LIN {X 0,Y 274.627,Z 437.441,A -85,B 0,C 180,E1 -17711.091,E2 -17711.091} C_VEL
LIN {X 0,Y 272.155,Z 443.733,A -85,B 0,C 180,E1 -17713.497,E2 -17713.497} C_VEL
LIN {X 0,Y 270.137,Z 449.54,A -85,B 0,C 180,E1 -17716.459,E2 -17716.459} C_VEL
LIN {X 0,Y 269.337,Z 451.749,A -85,B 0,C 180,E1 -17717.951,E2 -17717.951} C_VEL
LIN {X 0,Y 268.643,Z 455.017,A -85,B 0,C 180,E1 -17720.969,E2 -17720.969} C_VEL
LIN {X 0,Y 268.592,Z 456.649,A -85,B 0,C 180,E1 -17723.992,E2 -17723.992} C_VEL
LIN {X 0,Y 268.676,Z 456.883,A -85,B 0,C 180,E1 -17725.499,E2 -17725.499} C_VEL
LIN {X 0,Y 268.958,Z 456.687,A -85,B 0,C 180,E1 -17727.004,E2 -17727.004} C_VEL
LIN {X 0,Y 269.249,Z 456.062,A -85,B 0,C 180,E1 -17728.504,E2 -17728.504} C_VEL
LIN {X 0,Y 269.5,Z 453.773,A -85,B 0,C 180,E1 -17731.214,E2 -17731.214} C_VEL
LIN {X 0,Y 269.104,Z 455.004,A -85,B 0,C 180,E1 -17732.994,E2 -17732.994} C_VEL
LIN {X 0,Y 268.764,Z 455.392,A -85,B 0,C 180,E1 -17734.499,E2 -17734.499} C_VEL
LIN {X 0,Y 268.716,Z 454.986,A -85,B 0,C 180,E1 -17736.344,E2 -17736.344} C_VEL
LIN {X 0,Y 268.741,Z 454.264,A -85,B 0,C 180,E1 -17737.513,E2 -17737.513} C_VEL
LIN {X 0,Y 269.089,Z 451.749,A -85,B 0,C 180,E1 -17739.774,E2 -17739.774} C_VEL
LIN {X 0,Y 269.857,Z 447.728,A -85,B 0,C 180,E1 -17742.026,E2 -17742.026} C_VEL
LIN {X 0,Y 270.951,Z 443.145,A -85,B 0,C 180,E1 -17743.882,E2 -17743.882} C_VEL
LIN {X 0,Y 272.382,Z 437.177,A -85,B 0,C 180,E1 -17745.719,E2 -17745.719} C_VEL
LIN {X 0,Y 274.136,Z 429.673,A -85,B 0,C 180,E1 -17747.532,E2 -17747.532} C_VEL
LIN {X 0,Y 276.003,Z 420.924,A -85,B 0,C 180,E1 -17749.133,E2 -17749.133} C_VEL
LIN {X 0,Y 277.817,Z 411.718,A -85,B 0,C 180,E1 -17750.439,E2 -17750.439} C_VEL
LIN {X 0,Y 278.918,Z 404.593,A -85,B 0,C 180,E1 -17751.255,E2 -17751.255} C_VEL
LIN {X 0,Y 278.981,Z 396.262,A -85,B 0,C 180,E1 -17752.202,E2 -17752.202} C_VEL
LIN {X 0,Y 278.566,Z 384.711,A -85,B 0,C 180,E1 -17753.315,E2 -17753.315} C_VEL
LIN {X 0,Y 278.989,Z 376.477,A -85,B 0,C 180,E1 -17755.047,E2 -17755.047} C_VEL
LIN {X 0,Y 279.925,Z 365.219,A -85,B 0,C 180,E1 -17757.799,E2 -17757.799} C_VEL
LIN {X 0,Y 281.461,Z 354.384,A -85,B 0,C 180,E1 -17761.019,E2 -17761.019} C_VEL
LIN {X 0,Y 282.099,Z 351.247,A -85,B 0,C 180,E1 -17762.105,E2 -17762.105} C_VEL
LIN {X 0,Y 282.162,Z 348.83,A -85,B 0,C 180,E1 -17763.228,E2 -17763.228} C_VEL
LIN {X 0,Y 281.757,Z 343.357,A -85,B 0,C 180,E1 -17766.773,E2 -17766.773} C_VEL
LIN {X 0,Y 281.788,Z 340.66,A -85,B 0,C 180,E1 -17769.359,E2 -17769.359} C_VEL
LIN {X 0,Y 281.455,Z 339.512,A -85,B 0,C 180,E1 -17771.485,E2 -17771.485} C_VEL
LIN {X 0,Y 280.869,Z 339.07,A -85,B 0,C 180,E1 -17774.477,E2 -17774.477} C_VEL
LIN {X 0,Y 280.547,Z 339.568,A -85,B 0,C 180,E1 -17777.437,E2 -17777.437} C_VEL
LIN {X 0,Y 280.361,Z 341.176,A -85,B 0,C 180,E1 -17780.996,E2 -17780.996} C_VEL
LIN {X 0,Y 280.328,Z 342.758,A -85,B 0,C 180,E1 -17783.347,E2 -17783.347} C_VEL
LIN {X 0,Y 280.314,Z 345.504,A -85,B 0,C 180,E1 -17786.523,E2 -17786.523} C_VEL
LIN {X 0,Y 280,Z 347.801,A -85,B 0,C 180,E1 -17788.584,E2 -17788.584} C_VEL
LIN {X 0,Y 278.655,Z 352.411,A -85,B 0,C 180,E1 -17791.975,E2 -17791.975} C_VEL
LIN {X 0,Y 277.206,Z 359.26,A -85,B 0,C 180,E1 -17796.52,E2 -17796.52} C_VEL
LIN {X 0,Y 280.532,Z 368.404,A -85,B 0,C 180,E1 -17798.417,E2 -17798.417} C_VEL
LIN {X 0,Y 282.405,Z 375.568,A -85,B 0,C 180,E1 -17799.939,E2 -17799.939} C_VEL
LIN {X 0,Y 283.424,Z 383.27,A -85,B 0,C 180,E1 -17801.64,E2 -17801.64} C_VEL
LIN {X 0,Y 283.345,Z 385.026,A -85,B 0,C 180,E1 -17802.029,E2 -17802.029} C_VEL
LIN {X 0,Y 281.444,Z 391.557,A -85,B 0,C 180,E1 -17803.31,E2 -17803.31} C_VEL
LIN {X 0,Y 279.479,Z 397.018,A -85,B 0,C 180,E1 -17804.688,E2 -17804.688} C_VEL
LIN {X 0,Y 277.786,Z 401.348,A -85,B 0,C 180,E1 -17806.091,E2 -17806.091} C_VEL
LIN {X 0,Y 276.26,Z 404.765,A -85,B 0,C 180,E1 -17807.51,E2 -17807.51} C_VEL
LIN {X 0,Y 274.822,Z 407.385,A -85,B 0,C 180,E1 -17808.941,E2 -17808.941} C_VEL
LIN {X 0,Y 272.891,Z 409.903,A -85,B 0,C 180,E1 -17811.109,E2 -17811.109} C_VEL
LIN {X 0,Y 271.698,Z 410.764,A -85,B 0,C 180,E1 -17812.567,E2 -17812.567} C_VEL
LIN {X 0,Y 270.742,Z 410.941,A -85,B 0,C 180,E1 -17814.038,E2 -17814.038} C_VEL
LIN {X 0,Y 269.976,Z 410.449,A -85,B 0,C 180,E1 -17815.519,E2 -17815.519} C_VEL
LIN {X 0,Y 269.464,Z 409.29,A -85,B 0,C 180,E1 -17817.008,E2 -17817.008} C_VEL
LIN {X 0,Y 269.106,Z 407.446,A -85,B 0,C 180,E1 -17818.502,E2 -17818.502} C_VEL
LIN {X 0,Y 268.871,Z 404.869,A -85,B 0,C 180,E1 -17819.998,E2 -17819.998} C_VEL
LIN {X 0,Y 268.795,Z 399.475,A -85,B 0,C 180,E1 -17822.246,E2 -17822.246} C_VEL
LIN {X 0,Y 268.98,Z 393.345,A -85,B 0,C 180,E1 -17824.118,E2 -17824.118} C_VEL
LIN {X 0,Y 269.331,Z 387.173,A -85,B 0,C 180,E1 -17825.614,E2 -17825.614} C_VEL
LIN {X 0,Y 269.438,Z 379.922,A -85,B 0,C 180,E1 -17827.002,E2 -17827.002} C_VEL
LIN {X 0,Y 269.701,Z 371.818,A -85,B 0,C 180,E1 -17828.237,E2 -17828.237} C_VEL
LIN {X 0,Y 269.971,Z 362.059,A -85,B 0,C 180,E1 -17829.362,E2 -17829.362} C_VEL
LIN {X 0,Y 270.01,Z 354.616,A -85,B 0,C 180,E1 -17830.022,E2 -17830.022} C_VEL
LIN {X 0,Y 269.568,Z 350.628,A -85,B 0,C 180,E1 -17830.323,E2 -17830.323} C_VEL
LIN {X 0,Y 269.612,Z 340.781,A -85,B 0,C 180,E1 -17835.108,E2 -17835.108} C_VEL
LIN {X 0,Y 269.785,Z 331.31,A -85,B 0,C 180,E1 -17839.793,E2 -17839.793} C_VEL
LIN {X 0,Y 269.969,Z 323.565,A -85,B 0,C 180,E1 -17843.675,E2 -17843.675} C_VEL
LIN {X 0,Y 270.234,Z 316.909,A -85,B 0,C 180,E1 -17847.043,E2 -17847.043} C_VEL
LIN {X 0,Y 270.457,Z 310.793,A -85,B 0,C 180,E1 -17850.217,E2 -17850.217} C_VEL
LIN {X 0,Y 270.194,Z 310.826,A -85,B 0,C 180,E1 -17854.904,E2 -17854.904} C_VEL
LIN {X 0,Y 270.192,Z 310.828,A -85,B 0,C 180,E1 -17858.708,E2 -17858.708} C_VEL
LIN {X 0,Y 270.15,Z 310.834,A -85,B 0,C 180,E1 -17863.245,E2 -17863.245} C_VEL
LIN {X 0,Y 270.164,Z 310.831,A -85,B 0,C 180,E1 -17867.44,E2 -17867.44} C_VEL
LIN {X 0,Y 270.199,Z 310.825,A -85,B 0,C 180,E1 -17871.373,E2 -17871.373} C_VEL
LIN {X 0,Y 270.193,Z 310.828,A -85,B 0,C 180,E1 -17875.093,E2 -17875.093} C_VEL
LIN {X 0,Y 270.191,Z 310.826,A -85,B 0,C 180,E1 -17879.129,E2 -17879.129} C_VEL
LIN {X 0,Y 270.255,Z 310.819,A -85,B 0,C 180,E1 -17882.144,E2 -17882.144} C_VEL
LIN {X 0,Y 270.267,Z 310.817,A -85,B 0,C 180,E1 -17885.518,E2 -17885.518} C_VEL
LIN {X 0,Y 270.292,Z 310.816,A -85,B 0,C 180,E1 -17890.244,E2 -17890.244} C_VEL
LIN {X 0,Y 270.392,Z 310.801,A -85,B 0,C 180,E1 -17894.935,E2 -17894.935} C_VEL
LIN {X 0,Y 270.399,Z 310.8,A -85,B 0,C 180,E1 -17899.517,E2 -17899.517} C_VEL
LIN {X 0,Y 270.551,Z 310.783,A -85,B 0,C 180,E1 -17902.537,E2 -17902.537} C_VEL
LIN {X 0,Y 270.758,Z 310.757,A -85,B 0,C 180,E1 -17908.513,E2 -17908.513} C_VEL
LIN {X 0,Y 270.758,Z 310.757,A -85,B 0,C 180,E1 -17911.487,E2 -17911.487} C_VEL
LIN {X 0,Y 270.551,Z 310.783,A -85,B 0,C 180,E1 -17917.463,E2 -17917.463} C_VEL
LIN {X 0,Y 270.399,Z 310.8,A -85,B 0,C 180,E1 -17920.483,E2 -17920.483} C_VEL
LIN {X 0,Y 270.392,Z 310.801,A -85,B 0,C 180,E1 -17925.065,E2 -17925.065} C_VEL
LIN {X 0,Y 270.292,Z 310.816,A -85,B 0,C 180,E1 -17929.756,E2 -17929.756} C_VEL
LIN {X 0,Y 270.264,Z 310.817,A -85,B 0,C 180,E1 -17934.587,E2 -17934.587} C_VEL
LIN {X 0,Y 270.263,Z 310.818,A -85,B 0,C 180,E1 -17937.91,E2 -17937.91} C_VEL
LIN {X 0,Y 270.175,Z 310.832,A -85,B 0,C 180,E1 -17941.35,E2 -17941.35} C_VEL
LIN {X 0,Y 270.193,Z 310.828,A -85,B 0,C 180,E1 -17944.907,E2 -17944.907} C_VEL
LIN {X 0,Y 270.189,Z 310.827,A -85,B 0,C 180,E1 -17948.712,E2 -17948.712} C_VEL
LIN {X 0,Y 270.164,Z 310.831,A -85,B 0,C 180,E1 -17952.56,E2 -17952.56} C_VEL
LIN {X 0,Y 270.15,Z 310.834,A -85,B 0,C 180,E1 -17956.755,E2 -17956.755} C_VEL
LIN {X 0,Y 270.201,Z 310.826,A -85,B 0,C 180,E1 -17961.376,E2 -17961.376} C_VEL
LIN {X 0,Y 270.209,Z 310.824,A -85,B 0,C 180,E1 -17965.098,E2 -17965.098} C_VEL
LIN {X 0,Y 270.454,Z 310.901,A -85,B 0,C 180,E1 -17968.143,E2 -17968.143} C_VEL
LIN {X 0,Y 270.585,Z 313.036,A -85,B 0,C 180,E1 -17969.71,E2 -17969.71} C_VEL
LIN {X 0,Y 270.086,Z 318.744,A -85,B 0,C 180,E1 -17973.748,E2 -17973.748} C_VEL
LIN {X 0,Y 269.634,Z 324.585,A -85,B 0,C 180,E1 -17977.796,E2 -17977.796} C_VEL
LIN {X 0,Y 269.269,Z 330.42,A -85,B 0,C 180,E1 -17981.75,E2 -17981.75} C_VEL
LIN {X 0,Y 269.046,Z 335.5,A -85,B 0,C 180,E1 -17985.131,E2 -17985.131} C_VEL
LIN {X 0,Y 268.959,Z 338.816,A -85,B 0,C 180,E1 -17987.313,E2 -17987.313} C_VEL
LIN {X 0,Y 270.03,Z 351.262,A -85,B 0,C 180,E1 -17988.365,E2 -17988.365} C_VEL
LIN {X 0,Y 270.614,Z 358.543,A -85,B 0,C 180,E1 -17989.149,E2 -17989.149} C_VEL
LIN {X 0,Y 270.17,Z 368.515,A -85,B 0,C 180,E1 -17990.456,E2 -17990.456} C_VEL
LIN {X 0,Y 269.696,Z 378.68,A -85,B 0,C 180,E1 -17992.143,E2 -17992.143} C_VEL
LIN {X 0,Y 269.429,Z 387.587,A -85,B 0,C 180,E1 -17994.013,E2 -17994.013} C_VEL
LIN {X 0,Y 269.006,Z 394.618,A -85,B 0,C 180,E1 -17995.882,E2 -17995.882} C_VEL
LIN {X 0,Y 268.81,Z 400.158,A -85,B 0,C 180,E1 -17997.754,E2 -17997.754} C_VEL
LIN {X 0,Y 268.894,Z 405.229,A -85,B 0,C 180,E1 -18000.002,E2 -18000.002} C_VEL
LIN {X 0,Y 269.118,Z 407.757,A -85,B 0,C 180,E1 -18001.498,E2 -18001.498} C_VEL
LIN {X 0,Y 269.492,Z 409.646,A -85,B 0,C 180,E1 -18002.992,E2 -18002.992} C_VEL
LIN {X 0,Y 269.994,Z 410.901,A -85,B 0,C 180,E1 -18004.481,E2 -18004.481} C_VEL
LIN {X 0,Y 270.736,Z 411.555,A -85,B 0,C 180,E1 -18005.962,E2 -18005.962} C_VEL
LIN {X 0,Y 271.663,Z 411.63,A -85,B 0,C 180,E1 -18007.434,E2 -18007.434} C_VEL
LIN {X 0,Y 272.787,Z 411.119,A -85,B 0,C 180,E1 -18008.894,E2 -18008.894} C_VEL
LIN {X 0,Y 274.169,Z 409.989,A -85,B 0,C 180,E1 -18010.339,E2 -18010.339} C_VEL
LIN {X 0,Y 276.423,Z 407.237,A -85,B 0,C 180,E1 -18012.483,E2 -18012.483} C_VEL
LIN {X 0,Y 278.977,Z 403.105,A -85,B 0,C 180,E1 -18014.593,E2 -18014.593} C_VEL
LIN {X 0,Y 282.019,Z 397.428,A -85,B 0,C 180,E1 -18016.655,E2 -18016.655} C_VEL
LIN {X 0,Y 284.8,Z 391.401,A -85,B 0,C 180,E1 -18018.34,E2 -18018.34} C_VEL
LIN {X 0,Y 286.204,Z 387.731,A -85,B 0,C 180,E1 -18019.219,E2 -18019.219} C_VEL
LIN {X 0,Y 286.392,Z 384.84,A -85,B 0,C 180,E1 -18020.041,E2 -18020.041} C_VEL
LIN {X 0,Y 285.851,Z 381.836,A -85,B 0,C 180,E1 -18021.05,E2 -18021.05} C_VEL
LIN {X 0,Y 284.444,Z 379.4,A -85,B 0,C 180,E1 -18022.103,E2 -18022.103} C_VEL
LIN {X 0,Y 280.87,Z 375.089,A -85,B 0,C 180,E1 -18024.266,E2 -18024.266} C_VEL
LIN {X 0,Y 279.581,Z 372.512,A -85,B 0,C 180,E1 -18025.346,E2 -18025.346} C_VEL
LIN {X 0,Y 279.335,Z 371.508,A -85,B 0,C 180,E1 -18025.698,E2 -18025.698} C_VEL
LIN {X 0,Y 277.905,Z 365.619,A -85,B 0,C 180,E1 -18027.733,E2 -18027.733} C_VEL
LIN {X 0,Y 276.143,Z 359.405,A -85,B 0,C 180,E1 -18030.08,E2 -18030.08} C_VEL
LIN {X 0,Y 274.272,Z 354.936,A -85,B 0,C 180,E1 -18032.263,E2 -18032.263} C_VEL
LIN {X 0,Y 271.972,Z 350.628,A -85,B 0,C 180,E1 -18035.212,E2 -18035.212} C_VEL
LIN {X 0,Y 272.298,Z 350.182,A -85,B 0,C 180,E1 -18038.277,E2 -18038.277} C_VEL
LIN {X 0,Y 272.725,Z 350.677,A -85,B 0,C 180,E1 -18042.07,E2 -18042.07} C_VEL
LIN {X 0,Y 273.308,Z 352.228,A -85,B 0,C 180,E1 -18046.057,E2 -18046.057} C_VEL
LIN {X 0,Y 273.67,Z 353.475,A -85,B 0,C 180,E1 -18048.139,E2 -18048.139} C_VEL
LIN {X 0,Y 274.21,Z 355.799,A -85,B 0,C 180,E1 -18051.013,E2 -18051.013} C_VEL
LIN {X 0,Y 276.582,Z 360.694,A -85,B 0,C 180,E1 -18053.132,E2 -18053.132} C_VEL
LIN {X 0,Y 277.915,Z 362.494,A -85,B 0,C 180,E1 -18054.023,E2 -18054.023} C_VEL
LIN {X 0,Y 280.357,Z 367.956,A -85,B 0,C 180,E1 -18055.819,E2 -18055.819} C_VEL
LIN {X 0,Y 281.315,Z 375.382,A -85,B 0,C 180,E1 -18057.33,E2 -18057.33} C_VEL
LIN {X 0,Y 281.948,Z 387.904,A -85,B 0,C 180,E1 -18059.673,E2 -18059.673} C_VEL
LIN {X 0,Y 281.361,Z 398.895,A -85,B 0,C 180,E1 -18061.667,E2 -18061.667} C_VEL
LIN {X 0,Y 280.008,Z 406.994,A -85,B 0,C 180,E1 -18063.141,E2 -18063.141} C_VEL
LIN {X 0,Y 277.073,Z 416.211,A -85,B 0,C 180,E1 -18064.858,E2 -18064.858} C_VEL
LIN {X 0,Y 273.168,Z 425.604,A -85,B 0,C 180,E1 -18066.899,E2 -18066.899} C_VEL
LIN {X 0,Y 269.446,Z 434.425,A -85,B 0,C 180,E1 -18069.383,E2 -18069.383} C_VEL
LIN {X 0,Y 266.822,Z 440.501,A -85,B 0,C 180,E1 -18071.574,E2 -18071.574} C_VEL
LIN {X 0,Y 264.744,Z 445.446,A -85,B 0,C 180,E1 -18073.815,E2 -18073.815} C_VEL
LIN {X 0,Y 263.209,Z 449.382,A -85,B 0,C 180,E1 -18076.095,E2 -18076.095} C_VEL
LIN {X 0,Y 262.355,Z 451.48,A -85,B 0,C 180,E1 -18077.625,E2 -18077.625} C_VEL
LIN {X 0,Y 261.878,Z 453.174,A -85,B 0,C 180,E1 -18079.172,E2 -18079.172} C_VEL
LIN {X 0,Y 261.468,Z 455.364,A -85,B 0,C 180,E1 -18082.276,E2 -18082.276} C_VEL
LIN {X 0,Y 261.524,Z 455.905,A -85,B 0,C 180,E1 -18083.898,E2 -18083.898} C_VEL
LIN {X 0,Y 261.93,Z 455.684,A -85,B 0,C 180,E1 -18086.924,E2 -18086.924} C_VEL
LIN {X 0,Y 262.22,Z 454.979,A -85,B 0,C 180,E1 -18088.464,E2 -18088.464} C_VEL
LIN {X 0,Y 262.489,Z 452.482,A -85,B 0,C 180,E1 -18091.342,E2 -18091.342} C_VEL
LIN {X 0,Y 262.061,Z 453.944,A -85,B 0,C 180,E1 -18093.075,E2 -18093.075} C_VEL
LIN {X 0,Y 261.707,Z 454.505,A -85,B 0,C 180,E1 -18094.621,E2 -18094.621} C_VEL
LIN {X 0,Y 261.643,Z 454.408,A -85,B 0,C 180,E1 -18096.342,E2 -18096.342} C_VEL
LIN {X 0,Y 261.673,Z 453.757,A -85,B 0,C 180,E1 -18097.718,E2 -18097.718} C_VEL
LIN {X 0,Y 261.867,Z 452.442,A -85,B 0,C 180,E1 -18099.267,E2 -18099.267} C_VEL
LIN {X 0,Y 262.544,Z 449.245,A -85,B 0,C 180,E1 -18101.582,E2 -18101.582} C_VEL
LIN {X 0,Y 263.81,Z 444.596,A -85,B 0,C 180,E1 -18103.873,E2 -18103.873} C_VEL
LIN {X 0,Y 265.334,Z 439.323,A -85,B 0,C 180,E1 -18105.753,E2 -18105.753} C_VEL
LIN {X 0,Y 267.141,Z 432.669,A -85,B 0,C 180,E1 -18107.611,E2 -18107.611} C_VEL
LIN {X 0,Y 268.843,Z 425.988,A -85,B 0,C 180,E1 -18109.073,E2 -18109.073} C_VEL
LIN {X 0,Y 270.849,Z 417.563,A -85,B 0,C 180,E1 -18110.554,E2 -18110.554} C_VEL
LIN {X 0,Y 273.031,Z 407.211,A -85,B 0,C 180,E1 -18111.916,E2 -18111.916} C_VEL
LIN {X 0,Y 273.478,Z 399.542,A -85,B 0,C 180,E1 -18112.873,E2 -18112.873} C_VEL
LIN {X 0,Y 273.454,Z 389.243,A -85,B 0,C 180,E1 -18113.979,E2 -18113.979} C_VEL
LIN {X 0,Y 272.985,Z 384.727,A -85,B 0,C 180,E1 -18114.49,E2 -18114.49} C_VEL
LIN {X 0,Y 272.99,Z 382.104,A -85,B 0,C 180,E1 -18114.984,E2 -18114.984} C_VEL
LIN {X 0,Y 273.814,Z 371.617,A -85,B 0,C 180,E1 -18117.517,E2 -18117.517} C_VEL
LIN {X 0,Y 274.669,Z 364.395,A -85,B 0,C 180,E1 -18119.543,E2 -18119.543} C_VEL
LIN {X 0,Y 276.389,Z 355.842,A -85,B 0,C 180,E1 -18122.275,E2 -18122.275} C_VEL
LIN {X 0,Y 276.664,Z 353.951,A -85,B 0,C 180,E1 -18123.038,E2 -18123.038} C_VEL
LIN {X 0,Y 276.274,Z 349.326,A -85,B 0,C 180,E1 -18125.809,E2 -18125.809} C_VEL
LIN {X 0,Y 276.236,Z 346.589,A -85,B 0,C 180,E1 -18127.933,E2 -18127.933} C_VEL
LIN {X 0,Y 276.251,Z 345.028,A -85,B 0,C 180,E1 -18129.496,E2 -18129.496} C_VEL
LIN {X 0,Y 275.684,Z 343.649,A -85,B 0,C 180,E1 -18132.326,E2 -18132.326} C_VEL
LIN {X 0,Y 274.998,Z 343.398,A -85,B 0,C 180,E1 -18135.691,E2 -18135.691} C_VEL
LIN {X 0,Y 274.647,Z 343.941,A -85,B 0,C 180,E1 -18138.291,E2 -18138.291} C_VEL
LIN {X 0,Y 274.473,Z 344.699,A -85,B 0,C 180,E1 -18140.196,E2 -18140.196} C_VEL
LIN {X 0,Y 274.273,Z 346.957,A -85,B 0,C 180,E1 -18143.887,E2 -18143.887} C_VEL
LIN {X 0,Y 274.214,Z 348.388,A -85,B 0,C 180,E1 -18145.675,E2 -18145.675} C_VEL
LIN {X 0,Y 273.872,Z 350.567,A -85,B 0,C 180,E1 -18147.869,E2 -18147.869} C_VEL
LIN {X 0,Y 272.818,Z 354.086,A -85,B 0,C 180,E1 -18150.693,E2 -18150.693} C_VEL
LIN {X 0,Y 271.187,Z 360.381,A -85,B 0,C 180,E1 -18155.101,E2 -18155.101} C_VEL
LIN {X 0,Y 274.516,Z 369.396,A -85,B 0,C 180,E1 -18157.169,E2 -18157.169} C_VEL
LIN {X 0,Y 276.38,Z 376.908,A -85,B 0,C 180,E1 -18158.902,E2 -18158.902} C_VEL
LIN {X 0,Y 277.43,Z 384.794,A -85,B 0,C 180,E1 -18160.771,E2 -18160.771} C_VEL
LIN {X 0,Y 277.232,Z 387.906,A -85,B 0,C 180,E1 -18161.484,E2 -18161.484} C_VEL
LIN {X 0,Y 274.972,Z 394.379,A -85,B 0,C 180,E1 -18162.905,E2 -18162.905} C_VEL
LIN {X 0,Y 272.487,Z 400.55,A -85,B 0,C 180,E1 -18164.669,E2 -18164.669} C_VEL
LIN {X 0,Y 270.332,Z 405.102,A -85,B 0,C 180,E1 -18166.467,E2 -18166.467} C_VEL
LIN {X 0,Y 268.762,Z 407.845,A -85,B 0,C 180,E1 -18167.923,E2 -18167.923} C_VEL
LIN {X 0,Y 267.337,Z 409.835,A -85,B 0,C 180,E1 -18169.394,E2 -18169.394} C_VEL
LIN {X 0,Y 265.977,Z 411.136,A -85,B 0,C 180,E1 -18170.876,E2 -18170.876} C_VEL
LIN {X 0,Y 264.729,Z 411.773,A -85,B 0,C 180,E1 -18172.37,E2 -18172.37} C_VEL
LIN {X 0,Y 263.741,Z 411.735,A -85,B 0,C 180,E1 -18173.879,E2 -18173.879} C_VEL
LIN {X 0,Y 262.933,Z 411.022,A -85,B 0,C 180,E1 -18175.399,E2 -18175.399} C_VEL
LIN {X 0,Y 262.2,Z 408.665,A -85,B 0,C 180,E1 -18177.694,E2 -18177.694} C_VEL
LIN {X 0,Y 261.77,Z 404.748,A -85,B 0,C 180,E1 -18179.998,E2 -18179.998} C_VEL
LIN {X 0,Y 261.683,Z 400.142,A -85,B 0,C 180,E1 -18181.922,E2 -18181.922} C_VEL
LIN {X 0,Y 261.855,Z 393.952,A -85,B 0,C 180,E1 -18183.845,E2 -18183.845} C_VEL
LIN {X 0,Y 262.19,Z 387.737,A -85,B 0,C 180,E1 -18185.381,E2 -18185.381} C_VEL
LIN {X 0,Y 262.357,Z 380.386,A -85,B 0,C 180,E1 -18186.813,E2 -18186.813} C_VEL
LIN {X 0,Y 262.629,Z 371.489,A -85,B 0,C 180,E1 -18188.192,E2 -18188.192} C_VEL
LIN {X 0,Y 262.939,Z 360.827,A -85,B 0,C 180,E1 -18189.42,E2 -18189.42} C_VEL
LIN {X 0,Y 262.828,Z 354.006,A -85,B 0,C 180,E1 -18190.007,E2 -18190.007} C_VEL
LIN {X 0,Y 262.523,Z 351.276,A -85,B 0,C 180,E1 -18190.214,E2 -18190.214} C_VEL
LIN {X 0,Y 262.518,Z 342.111,A -85,B 0,C 180,E1 -18194.716,E2 -18194.716} C_VEL
LIN {X 0,Y 262.702,Z 332.471,A -85,B 0,C 180,E1 -18199.534,E2 -18199.534} C_VEL
LIN {X 0,Y 262.903,Z 324.362,A -85,B 0,C 180,E1 -18203.637,E2 -18203.637} C_VEL
LIN {X 0,Y 263.198,Z 316.592,A -85,B 0,C 180,E1 -18207.61,E2 -18207.61} C_VEL
LIN {X 0,Y 263.407,Z 311.672,A -85,B 0,C 180,E1 -18210.126,E2 -18210.126} C_VEL
LIN {X 0,Y 263.169,Z 311.699,A -85,B 0,C 180,E1 -18214.12,E2 -18214.12} C_VEL
LIN {X 0,Y 263.151,Z 311.704,A -85,B 0,C 180,E1 -18217.895,E2 -18217.895} C_VEL
LIN {X 0,Y 263.103,Z 311.708,A -85,B 0,C 180,E1 -18221.894,E2 -18221.894} C_VEL
LIN {X 0,Y 263.098,Z 311.71,A -85,B 0,C 180,E1 -18226.153,E2 -18226.153} C_VEL
LIN {X 0,Y 263.098,Z 311.709,A -85,B 0,C 180,E1 -18230.126,E2 -18230.126} C_VEL
LIN {X 0,Y 263.155,Z 311.703,A -85,B 0,C 180,E1 -18234.017,E2 -18234.017} C_VEL
LIN {X 0,Y 263.124,Z 311.706,A -85,B 0,C 180,E1 -18237.71,E2 -18237.71} C_VEL
LIN {X 0,Y 263.192,Z 311.698,A -85,B 0,C 180,E1 -18241.782,E2 -18241.782} C_VEL
LIN {X 0,Y 263.216,Z 311.696,A -85,B 0,C 180,E1 -18245.199,E2 -18245.199} C_VEL
LIN {X 0,Y 263.254,Z 311.689,A -85,B 0,C 180,E1 -18249.693,E2 -18249.693} C_VEL
LIN {X 0,Y 263.34,Z 311.682,A -85,B 0,C 180,E1 -18254.521,E2 -18254.521} C_VEL
LIN {X 0,Y 263.338,Z 311.679,A -85,B 0,C 180,E1 -18259.233,E2 -18259.233} C_VEL
LIN {X 0,Y 263.515,Z 311.661,A -85,B 0,C 180,E1 -18262.337,E2 -18262.337} C_VEL
LIN {X 0,Y 263.722,Z 311.634,A -85,B 0,C 180,E1 -18268.473,E2 -18268.473} C_VEL
LIN {X 0,Y 263.722,Z 311.634,A -85,B 0,C 180,E1 -18271.527,E2 -18271.527} C_VEL
LIN {X 0,Y 263.515,Z 311.661,A -85,B 0,C 180,E1 -18277.663,E2 -18277.663} C_VEL
LIN {X 0,Y 263.338,Z 311.679,A -85,B 0,C 180,E1 -18280.767,E2 -18280.767} C_VEL
LIN {X 0,Y 263.34,Z 311.682,A -85,B 0,C 180,E1 -18285.479,E2 -18285.479} C_VEL
LIN {X 0,Y 263.258,Z 311.689,A -85,B 0,C 180,E1 -18290.307,E2 -18290.307} C_VEL
LIN {X 0,Y 263.199,Z 311.701,A -85,B 0,C 180,E1 -18295.292,E2 -18295.292} C_VEL
LIN {X 0,Y 263.17,Z 311.701,A -85,B 0,C 180,E1 -18298.731,E2 -18298.731} C_VEL
LIN {X 0,Y 263.124,Z 311.706,A -85,B 0,C 180,E1 -18302.29,E2 -18302.29} C_VEL
LIN {X 0,Y 263.175,Z 311.702,A -85,B 0,C 180,E1 -18306.765,E2 -18306.765} C_VEL
LIN {X 0,Y 263.117,Z 311.709,A -85,B 0,C 180,E1 -18311.595,E2 -18311.595} C_VEL
LIN {X 0,Y 263.094,Z 311.709,A -85,B 0,C 180,E1 -18316.013,E2 -18316.013} C_VEL
LIN {X 0,Y 263.085,Z 311.712,A -85,B 0,C 180,E1 -18320.127,E2 -18320.127} C_VEL
LIN {X 0,Y 263.156,Z 311.702,A -85,B 0,C 180,E1 -18324.02,E2 -18324.02} C_VEL
LIN {X 0,Y 263.404,Z 311.753,A -85,B 0,C 180,E1 -18328.105,E2 -18328.105} C_VEL
LIN {X 0,Y 263.477,Z 314.888,A -85,B 0,C 180,E1 -18330.434,E2 -18330.434} C_VEL
LIN {X 0,Y 262.916,Z 320.809,A -85,B 0,C 180,E1 -18334.681,E2 -18334.681} C_VEL
LIN {X 0,Y 262.5,Z 326.69,A -85,B 0,C 180,E1 -18338.815,E2 -18338.815} C_VEL
LIN {X 0,Y 262.117,Z 332.563,A -85,B 0,C 180,E1 -18342.849,E2 -18342.849} C_VEL
LIN {X 0,Y 261.875,Z 339.108,A -85,B 0,C 180,E1 -18347.26,E2 -18347.26} C_VEL
LIN {X 0,Y 263.018,Z 352.365,A -85,B 0,C 180,E1 -18348.442,E2 -18348.442} C_VEL
LIN {X 0,Y 263.534,Z 359.522,A -85,B 0,C 180,E1 -18349.243,E2 -18349.243} C_VEL
LIN {X 0,Y 263.026,Z 370.656,A -85,B 0,C 180,E1 -18350.777,E2 -18350.777} C_VEL
LIN {X 0,Y 262.467,Z 380.858,A -85,B 0,C 180,E1 -18352.576,E2 -18352.576} C_VEL
LIN {X 0,Y 262.309,Z 388.314,A -85,B 0,C 180,E1 -18354.236,E2 -18354.236} C_VEL
LIN {X 0,Y 261.872,Z 395.282,A -85,B 0,C 180,E1 -18356.155,E2 -18356.155} C_VEL
LIN {X 0,Y 261.706,Z 401.832,A -85,B 0,C 180,E1 -18358.463,E2 -18358.463} C_VEL
LIN {X 0,Y 261.953,Z 406.669,A -85,B 0,C 180,E1 -18360.771,E2 -18360.771} C_VEL
LIN {X 0,Y 262.438,Z 409.974,A -85,B 0,C 180,E1 -18363.072,E2 -18363.072} C_VEL
LIN {X 0,Y 262.951,Z 411.434,A -85,B 0,C 180,E1 -18364.601,E2 -18364.601} C_VEL
LIN {X 0,Y 263.736,Z 412.299,A -85,B 0,C 180,E1 -18366.121,E2 -18366.121} C_VEL
LIN {X 0,Y 264.683,Z 412.546,A -85,B 0,C 180,E1 -18367.631,E2 -18367.631} C_VEL
LIN {X 0,Y 265.858,Z 412.223,A -85,B 0,C 180,E1 -18369.128,E2 -18369.128} C_VEL
LIN {X 0,Y 267.307,Z 411.326,A -85,B 0,C 180,E1 -18370.607,E2 -18370.607} C_VEL
LIN {X 0,Y 269.671,Z 408.895,A -85,B 0,C 180,E1 -18372.8,E2 -18372.8} C_VEL
LIN {X 0,Y 272.36,Z 405.131,A -85,B 0,C 180,E1 -18374.956,E2 -18374.956} C_VEL
LIN {X 0,Y 275.535,Z 399.897,A -85,B 0,C 180,E1 -18377.059,E2 -18377.059} C_VEL
LIN {X 0,Y 278.385,Z 394.284,A -85,B 0,C 180,E1 -18378.778,E2 -18378.778} C_VEL
LIN {X 0,Y 280.234,Z 390.332,A -85,B 0,C 180,E1 -18379.791,E2 -18379.791} C_VEL
LIN {X 0,Y 280.649,Z 384.473,A -85,B 0,C 180,E1 -18381.616,E2 -18381.616} C_VEL
LIN {X 0,Y 280.195,Z 376.671,A -85,B 0,C 180,E1 -18384.032,E2 -18384.032} C_VEL
LIN {X 0,Y 279.335,Z 371.508,A -85,B 0,C 180,E1 -18385.698,E2 -18385.698} C_VEL
LIN {X 0,Y 278.305,Z 368.98,A -85,B 0,C 180,E1 -18386.771,E2 -18386.771} C_VEL
LIN {X 0,Y 276.634,Z 367.317,A -85,B 0,C 180,E1 -18387.898,E2 -18387.898} C_VEL
LIN {X 0,Y 272.881,Z 364.902,A -85,B 0,C 180,E1 -18390.232,E2 -18390.232} C_VEL
LIN {X 0,Y 271.505,Z 363.246,A -85,B 0,C 180,E1 -18391.415,E2 -18391.415} C_VEL
LIN {X 0,Y 271.21,Z 362.516,A -85,B 0,C 180,E1 -18391.804,E2 -18391.804} C_VEL
LIN {X 0,Y 270.011,Z 359.671,A -85,B 0,C 180,E1 -18393.6,E2 -18393.6} C_VEL
LIN {X 0,Y 268.801,Z 356.664,A -85,B 0,C 180,E1 -18395.853,E2 -18395.853} C_VEL
LIN {X 0,Y 267.173,Z 354.982,A -85,B 0,C 180,E1 -18399.15,E2 -18399.15} C_VEL
LIN {X 0,Y 266.859,Z 354.639,A -85,B 0,C 180,E1 -18401.18,E2 -18401.18} C_VEL
LIN {X 0,Y 266.952,Z 354.984,A -85,B 0,C 180,E1 -18403.198,E2 -18403.198} C_VEL
LIN {X 0,Y 267.458,Z 356.072,A -85,B 0,C 180,E1 -18405.195,E2 -18405.195} C_VEL
LIN {X 0,Y 268.964,Z 358.817,A -85,B 0,C 180,E1 -18408.119,E2 -18408.119} C_VEL
LIN {X 0,Y 270.747,Z 361.384,A -85,B 0,C 180,E1 -18410.166,E2 -18410.166} C_VEL
LIN {X 0,Y 274.796,Z 369.35,A -85,B 0,C 180,E1 -18413.968,E2 -18413.968} C_VEL
LIN {X 0,Y 276.202,Z 373.331,A -85,B 0,C 180,E1 -18415.279,E2 -18415.279} C_VEL
LIN {X 0,Y 276.724,Z 381.064,A -85,B 0,C 180,E1 -18416.943,E2 -18416.943} C_VEL
LIN {X 0,Y 276.609,Z 392.543,A -85,B 0,C 180,E1 -18419.236,E2 -18419.236} C_VEL
LIN {X 0,Y 275.632,Z 401.692,A -85,B 0,C 180,E1 -18421.023,E2 -18421.023} C_VEL
LIN {X 0,Y 273.994,Z 409.279,A -85,B 0,C 180,E1 -18422.503,E2 -18422.503} C_VEL
LIN {X 0,Y 270.797,Z 417.927,A -85,B 0,C 180,E1 -18424.233,E2 -18424.233} C_VEL
LIN {X 0,Y 266.767,Z 426.795,A -85,B 0,C 180,E1 -18426.311,E2 -18426.311} C_VEL
LIN {X 0,Y 262.852,Z 435.108,A -85,B 0,C 180,E1 -18428.841,E2 -18428.841} C_VEL
LIN {X 0,Y 259.64,Z 441.857,A -85,B 0,C 180,E1 -18431.518,E2 -18431.518} C_VEL
LIN {X 0,Y 257.323,Z 446.878,A -85,B 0,C 180,E1 -18434.15,E2 -18434.15} C_VEL
LIN {X 0,Y 256.298,Z 449.25,A -85,B 0,C 180,E1 -18435.712,E2 -18435.712} C_VEL
LIN {X 0,Y 255.389,Z 451.169,A -85,B 0,C 180,E1 -18437.282,E2 -18437.282} C_VEL
LIN {X 0,Y 254.55,Z 453.897,A -85,B 0,C 180,E1 -18440.465,E2 -18440.465} C_VEL
LIN {X 0,Y 254.445,Z 455.051,A -85,B 0,C 180,E1 -18443.657,E2 -18443.657} C_VEL
LIN {X 0,Y 254.898,Z 454.654,A -85,B 0,C 180,E1 -18446.839,E2 -18446.839} C_VEL
LIN {X 0,Y 255.207,Z 453.799,A -85,B 0,C 180,E1 -18448.422,E2 -18448.422} C_VEL
LIN {X 0,Y 255.521,Z 451.096,A -85,B 0,C 180,E1 -18451.379,E2 -18451.379} C_VEL
LIN {X 0,Y 255.038,Z 452.74,A -85,B 0,C 180,E1 -18453.159,E2 -18453.159} C_VEL
LIN {X 0,Y 254.692,Z 453.495,A -85,B 0,C 180,E1 -18454.749,E2 -18454.749} C_VEL
LIN {X 0,Y 254.591,Z 453.619,A -85,B 0,C 180,E1 -18456.38,E2 -18456.38} C_VEL
LIN {X 0,Y 254.616,Z 453.126,A -85,B 0,C 180,E1 -18457.933,E2 -18457.933} C_VEL
LIN {X 0,Y 254.83,Z 452.017,A -85,B 0,C 180,E1 -18459.525,E2 -18459.525} C_VEL
LIN {X 0,Y 255.571,Z 449.245,A -85,B 0,C 180,E1 -18461.902,E2 -18461.902} C_VEL
LIN {X 0,Y 256.921,Z 444.934,A -85,B 0,C 180,E1 -18464.252,E2 -18464.252} C_VEL
LIN {X 0,Y 258.881,Z 438.973,A -85,B 0,C 180,E1 -18466.562,E2 -18466.562} C_VEL
LIN {X 0,Y 260.908,Z 432.566,A -85,B 0,C 180,E1 -18468.452,E2 -18468.452} C_VEL
LIN {X 0,Y 262.818,Z 426.086,A -85,B 0,C 180,E1 -18469.935,E2 -18469.935} C_VEL
LIN {X 0,Y 265.216,Z 417.199,A -85,B 0,C 180,E1 -18471.568,E2 -18471.568} C_VEL
LIN {X 0,Y 267.271,Z 408.827,A -85,B 0,C 180,E1 -18472.725,E2 -18472.725} C_VEL
LIN {X 0,Y 267.963,Z 401.175,A -85,B 0,C 180,E1 -18473.76,E2 -18473.76} C_VEL
LIN {X 0,Y 268.276,Z 389.595,A -85,B 0,C 180,E1 -18475.117,E2 -18475.117} C_VEL
LIN {X 0,Y 267.23,Z 382.914,A -85,B 0,C 180,E1 -18476.057,E2 -18476.057} C_VEL
LIN {X 0,Y 268.287,Z 373.418,A -85,B 0,C 180,E1 -18478.458,E2 -18478.458} C_VEL
LIN {X 0,Y 269.84,Z 363.667,A -85,B 0,C 180,E1 -18481.393,E2 -18481.393} C_VEL
LIN {X 0,Y 270.921,Z 358.997,A -85,B 0,C 180,E1 -18483.009,E2 -18483.009} C_VEL
LIN {X 0,Y 271.009,Z 357.094,A -85,B 0,C 180,E1 -18483.914,E2 -18483.914} C_VEL
LIN {X 0,Y 270.728,Z 352.791,A -85,B 0,C 180,E1 -18486.661,E2 -18486.661} C_VEL
LIN {X 0,Y 270.66,Z 350.2,A -85,B 0,C 180,E1 -18488.83,E2 -18488.83} C_VEL
LIN {X 0,Y 270.375,Z 348.518,A -85,B 0,C 180,E1 -18491.076,E2 -18491.076} C_VEL
LIN {X 0,Y 269.832,Z 347.813,A -85,B 0,C 180,E1 -18493.171,E2 -18493.171} C_VEL
LIN {X 0,Y 269.359,Z 347.613,A -85,B 0,C 180,E1 -18495.211,E2 -18495.211} C_VEL
LIN {X 0,Y 268.988,Z 347.801,A -85,B 0,C 180,E1 -18497.208,E2 -18497.208} C_VEL
LIN {X 0,Y 268.471,Z 349.148,A -85,B 0,C 180,E1 -18501.076,E2 -18501.076} C_VEL
LIN {X 0,Y 268.198,Z 351.45,A -85,B 0,C 180,E1 -18504.793,E2 -18504.793} C_VEL
LIN {X 0,Y 267.859,Z 353.461,A -85,B 0,C 180,E1 -18507.099,E2 -18507.099} C_VEL
LIN {X 0,Y 266.827,Z 356.747,A -85,B 0,C 180,E1 -18509.969,E2 -18509.969} C_VEL
LIN {X 0,Y 265.324,Z 361.423,A -85,B 0,C 180,E1 -18513.5,E2 -18513.5} C_VEL
LIN {X 0,Y 268.617,Z 370.615,A -85,B 0,C 180,E1 -18515.836,E2 -18515.836} C_VEL
LIN {X 0,Y 270.732,Z 379.454,A -85,B 0,C 180,E1 -18518.054,E2 -18518.054} C_VEL
LIN {X 0,Y 271.494,Z 386.612,A -85,B 0,C 180,E1 -18519.916,E2 -18519.916} C_VEL
LIN {X 0,Y 271.405,Z 389.745,A -85,B 0,C 180,E1 -18520.727,E2 -18520.727} C_VEL
LIN {X 0,Y 268.547,Z 397.252,A -85,B 0,C 180,E1 -18522.483,E2 -18522.483} C_VEL
LIN {X 0,Y 266.427,Z 401.869,A -85,B 0,C 180,E1 -18523.918,E2 -18523.918} C_VEL
LIN {X 0,Y 263.669,Z 407.038,A -85,B 0,C 180,E1 -18526.118,E2 -18526.118} C_VEL
LIN {X 0,Y 262.004,Z 409.479,A -85,B 0,C 180,E1 -18527.607,E2 -18527.607} C_VEL
LIN {X 0,Y 260.505,Z 411.203,A -85,B 0,C 180,E1 -18529.112,E2 -18529.112} C_VEL
LIN {X 0,Y 259.052,Z 412.264,A -85,B 0,C 180,E1 -18530.63,E2 -18530.63} C_VEL
LIN {X 0,Y 257.749,Z 412.663,A -85,B 0,C 180,E1 -18532.162,E2 -18532.162} C_VEL
LIN {X 0,Y 256.725,Z 412.392,A -85,B 0,C 180,E1 -18533.711,E2 -18533.711} C_VEL
LIN {X 0,Y 255.894,Z 411.465,A -85,B 0,C 180,E1 -18535.272,E2 -18535.272} C_VEL
LIN {X 0,Y 255.121,Z 408.853,A -85,B 0,C 180,E1 -18537.63,E2 -18537.63} C_VEL
LIN {X 0,Y 254.671,Z 404.546,A -85,B 0,C 180,E1 -18539.998,E2 -18539.998} C_VEL
LIN {X 0,Y 254.597,Z 399.586,A -85,B 0,C 180,E1 -18541.975,E2 -18541.975} C_VEL
LIN {X 0,Y 254.789,Z 393.113,A -85,B 0,C 180,E1 -18543.952,E2 -18543.952} C_VEL
LIN {X 0,Y 255.149,Z 386.44,A -85,B 0,C 180,E1 -18545.53,E2 -18545.53} C_VEL
LIN {X 0,Y 255.311,Z 378.068,A -85,B 0,C 180,E1 -18547.1,E2 -18547.1} C_VEL
LIN {X 0,Y 255.593,Z 369.789,A -85,B 0,C 180,E1 -18548.297,E2 -18548.297} C_VEL
LIN {X 0,Y 255.859,Z 360.095,A -85,B 0,C 180,E1 -18549.384,E2 -18549.384} C_VEL
LIN {X 0,Y 255.736,Z 354.216,A -85,B 0,C 180,E1 -18549.888,E2 -18549.888} C_VEL
LIN {X 0,Y 255.478,Z 351.884,A -85,B 0,C 180,E1 -18550.098,E2 -18550.098} C_VEL
LIN {X 0,Y 255.454,Z 342.054,A -85,B 0,C 180,E1 -18554.994,E2 -18554.994} C_VEL
LIN {X 0,Y 255.669,Z 332.068,A -85,B 0,C 180,E1 -18560.059,E2 -18560.059} C_VEL
LIN {X 0,Y 255.917,Z 323.736,A -85,B 0,C 180,E1 -18564.324,E2 -18564.324} C_VEL
LIN {X 0,Y 256.194,Z 315.44,A -85,B 0,C 180,E1 -18568.617,E2 -18568.617} C_VEL
LIN {X 0,Y 256.359,Z 312.55,A -85,B 0,C 180,E1 -18570.132,E2 -18570.132} C_VEL
LIN {X 0,Y 256.101,Z 312.583,A -85,B 0,C 180,E1 -18575.187,E2 -18575.187} C_VEL
LIN {X 0,Y 256.06,Z 312.591,A -85,B 0,C 180,E1 -18579.141,E2 -18579.141} C_VEL
LIN {X 0,Y 256.037,Z 312.591,A -85,B 0,C 180,E1 -18583.329,E2 -18583.329} C_VEL
LIN {X 0,Y 256.062,Z 312.586,A -85,B 0,C 180,E1 -18587.818,E2 -18587.818} C_VEL
LIN {X 0,Y 256.064,Z 312.588,A -85,B 0,C 180,E1 -18590.856,E2 -18590.856} C_VEL
LIN {X 0,Y 256.123,Z 312.582,A -85,B 0,C 180,E1 -18592.866,E2 -18592.866} C_VEL
LIN {X 0,Y 256.059,Z 312.591,A -85,B 0,C 180,E1 -18596.706,E2 -18596.706} C_VEL
LIN {X 0,Y 256.105,Z 312.582,A -85,B 0,C 180,E1 -18600.399,E2 -18600.399} C_VEL
LIN {X 0,Y 256.179,Z 312.574,A -85,B 0,C 180,E1 -18604.86,E2 -18604.86} C_VEL
LIN {X 0,Y 256.159,Z 312.573,A -85,B 0,C 180,E1 -18609.104,E2 -18609.104} C_VEL
LIN {X 0,Y 256.29,Z 312.561,A -85,B 0,C 180,E1 -18614.084,E2 -18614.084} C_VEL
LIN {X 0,Y 256.28,Z 312.559,A -85,B 0,C 180,E1 -18618.933,E2 -18618.933} C_VEL
LIN {X 0,Y 256.479,Z 312.539,A -85,B 0,C 180,E1 -18622.125,E2 -18622.125} C_VEL
LIN {X 0,Y 256.442,Z 312.538,A -85,B 0,C 180,E1 -18626.858,E2 -18626.858} C_VEL
LIN {X 0,Y 256.684,Z 312.511,A -85,B 0,C 180,E1 -18628.431,E2 -18628.431} C_VEL
LIN {X 0,Y 256.685,Z 312.511,A -85,B 0,C 180,E1 -18631.569,E2 -18631.569} C_VEL
LIN {X 0,Y 256.444,Z 312.54,A -85,B 0,C 180,E1 -18636.294,E2 -18636.294} C_VEL
LIN {X 0,Y 256.416,Z 312.545,A -85,B 0,C 180,E1 -18639.465,E2 -18639.465} C_VEL
LIN {X 0,Y 256.244,Z 312.564,A -85,B 0,C 180,E1 -18644.291,E2 -18644.291} C_VEL
LIN {X 0,Y 256.2,Z 312.573,A -85,B 0,C 180,E1 -18647.563,E2 -18647.563} C_VEL
LIN {X 0,Y 256.175,Z 312.573,A -85,B 0,C 180,E1 -18651.137,E2 -18651.137} C_VEL
LIN {X 0,Y 256.179,Z 312.574,A -85,B 0,C 180,E1 -18655.14,E2 -18655.14} C_VEL
LIN {X 0,Y 256.105,Z 312.582,A -85,B 0,C 180,E1 -18659.601,E2 -18659.601} C_VEL
LIN {X 0,Y 256.059,Z 312.591,A -85,B 0,C 180,E1 -18663.294,E2 -18663.294} C_VEL
LIN {X 0,Y 256.107,Z 312.583,A -85,B 0,C 180,E1 -18667.273,E2 -18667.273} C_VEL
LIN {X 0,Y 256.047,Z 312.592,A -85,B 0,C 180,E1 -18671.205,E2 -18671.205} C_VEL
LIN {X 0,Y 256.033,Z 312.59,A -85,B 0,C 180,E1 -18675.536,E2 -18675.536} C_VEL
LIN {X 0,Y 256.034,Z 312.592,A -85,B 0,C 180,E1 -18678.796,E2 -18678.796} C_VEL
LIN {X 0,Y 256.12,Z 312.583,A -85,B 0,C 180,E1 -18682.869,E2 -18682.869} C_VEL
LIN {X 0,Y 256.374,Z 312.555,A -85,B 0,C 180,E1 -18688.039,E2 -18688.039} C_VEL
LIN {X 0,Y 256.409,Z 315.738,A -85,B 0,C 180,E1 -18690.441,E2 -18690.441} C_VEL
LIN {X 0,Y 255.79,Z 322.055,A -85,B 0,C 180,E1 -18695.053,E2 -18695.053} C_VEL
LIN {X 0,Y 255.381,Z 328.04,A -85,B 0,C 180,E1 -18699.337,E2 -18699.337} C_VEL
LIN {X 0,Y 254.945,Z 334.711,A -85,B 0,C 180,E1 -18704,E2 -18704} C_VEL
LIN {X 0,Y 254.799,Z 339.548,A -85,B 0,C 180,E1 -18707.254,E2 -18707.254} C_VEL
LIN {X 0,Y 255.806,Z 351.46,A -85,B 0,C 180,E1 -18708.312,E2 -18708.312} C_VEL
LIN {X 0,Y 256.453,Z 358.873,A -85,B 0,C 180,E1 -18709.142,E2 -18709.142} C_VEL
LIN {X 0,Y 255.939,Z 370.267,A -85,B 0,C 180,E1 -18710.738,E2 -18710.738} C_VEL
LIN {X 0,Y 255.445,Z 379.495,A -85,B 0,C 180,E1 -18712.37,E2 -18712.37} C_VEL
LIN {X 0,Y 255.261,Z 387.348,A -85,B 0,C 180,E1 -18714.076,E2 -18714.076} C_VEL
LIN {X 0,Y 254.806,Z 394.682,A -85,B 0,C 180,E1 -18716.048,E2 -18716.048} C_VEL
LIN {X 0,Y 254.618,Z 400.535,A -85,B 0,C 180,E1 -18718.025,E2 -18718.025} C_VEL
LIN {X 0,Y 254.695,Z 405.12,A -85,B 0,C 180,E1 -18720.002,E2 -18720.002} C_VEL
LIN {X 0,Y 255.139,Z 409.224,A -85,B 0,C 180,E1 -18722.37,E2 -18722.37} C_VEL
LIN {X 0,Y 255.911,Z 411.908,A -85,B 0,C 180,E1 -18724.728,E2 -18724.728} C_VEL
LIN {X 0,Y 256.721,Z 412.945,A -85,B 0,C 180,E1 -18726.289,E2 -18726.289} C_VEL
LIN {X 0,Y 257.703,Z 413.419,A -85,B 0,C 180,E1 -18727.839,E2 -18727.839} C_VEL
LIN {X 0,Y 258.931,Z 413.307,A -85,B 0,C 180,E1 -18729.375,E2 -18729.375} C_VEL
LIN {X 0,Y 260.446,Z 412.587,A -85,B 0,C 180,E1 -18730.89,E2 -18730.89} C_VEL
LIN {X 0,Y 262.018,Z 411.341,A -85,B 0,C 180,E1 -18732.393,E2 -18732.393} C_VEL
LIN {X 0,Y 264.765,Z 408.414,A -85,B 0,C 180,E1 -18734.608,E2 -18734.608} C_VEL
LIN {X 0,Y 267.878,Z 404.073,A -85,B 0,C 180,E1 -18736.776,E2 -18736.776} C_VEL
LIN {X 0,Y 271.42,Z 398.287,A -85,B 0,C 180,E1 -18738.887,E2 -18738.887} C_VEL
LIN {X 0,Y 274.013,Z 393.467,A -85,B 0,C 180,E1 -18740.26,E2 -18740.26} C_VEL
LIN {X 0,Y 274.598,Z 391.124,A -85,B 0,C 180,E1 -18740.998,E2 -18740.998} C_VEL
LIN {X 0,Y 275.006,Z 384.215,A -85,B 0,C 180,E1 -18743.337,E2 -18743.337} C_VEL
LIN {X 0,Y 274.516,Z 377.072,A -85,B 0,C 180,E1 -18745.801,E2 -18745.801} C_VEL
LIN {X 0,Y 273.405,Z 370.528,A -85,B 0,C 180,E1 -18748.23,E2 -18748.23} C_VEL
LIN {X 0,Y 272.123,Z 364.854,A -85,B 0,C 180,E1 -18750.572,E2 -18750.572} C_VEL
LIN {X 0,Y 271.21,Z 362.516,A -85,B 0,C 180,E1 -18751.804,E2 -18751.804} C_VEL
LIN {X 0,Y 270.593,Z 361.35,A -85,B 0,C 180,E1 -18752.586,E2 -18752.586} C_VEL
LIN {X 0,Y 269.216,Z 360.728,A -85,B 0,C 180,E1 -18753.8,E2 -18753.8} C_VEL
LIN {X 0,Y 264.987,Z 361.988,A -85,B 0,C 180,E1 -18757.586,E2 -18757.586} C_VEL
LIN {X 0,Y 264.561,Z 361.868,A -85,B 0,C 180,E1 -18758.458,E2 -18758.458} C_VEL
LIN {X 0,Y 264.28,Z 361.411,A -85,B 0,C 180,E1 -18759.662,E2 -18759.662} C_VEL
LIN {X 0,Y 264.125,Z 361.268,A -85,B 0,C 180,E1 -18761.837,E2 -18761.837} C_VEL
LIN {X 0,Y 264.426,Z 362.05,A -85,B 0,C 180,E1 -18764.142,E2 -18764.142} C_VEL
LIN {X 0,Y 265.223,Z 363.753,A -85,B 0,C 180,E1 -18766.452,E2 -18766.452} C_VEL
LIN {X 0,Y 267.395,Z 367.338,A -85,B 0,C 180,E1 -18769.662,E2 -18769.662} C_VEL
LIN {X 0,Y 268.472,Z 369.921,A -85,B 0,C 180,E1 -18771.077,E2 -18771.077} C_VEL
LIN {X 0,Y 270.914,Z 374.949,A -85,B 0,C 180,E1 -18773.535,E2 -18773.535} C_VEL
LIN {X 0,Y 271.829,Z 377.925,A -85,B 0,C 180,E1 -18774.585,E2 -18774.585} C_VEL
LIN {X 0,Y 271.924,Z 384.918,A -85,B 0,C 180,E1 -18776.205,E2 -18776.205} C_VEL
LIN {X 0,Y 271.311,Z 395.346,A -85,B 0,C 180,E1 -18778.449,E2 -18778.449} C_VEL
LIN {X 0,Y 269.9,Z 404.4,A -85,B 0,C 180,E1 -18780.347,E2 -18780.347} C_VEL
LIN {X 0,Y 267.98,Z 411.482,A -85,B 0,C 180,E1 -18781.831,E2 -18781.831} C_VEL
LIN {X 0,Y 264.554,Z 419.632,A -85,B 0,C 180,E1 -18783.578,E2 -18783.578} C_VEL
LIN {X 0,Y 260.382,Z 427.929,A -85,B 0,C 180,E1 -18785.694,E2 -18785.694} C_VEL
LIN {X 0,Y 256.294,Z 435.797,A -85,B 0,C 180,E1 -18788.272,E2 -18788.272} C_VEL
LIN {X 0,Y 252.755,Z 442.483,A -85,B 0,C 180,E1 -18791.166,E2 -18791.166} C_VEL
LIN {X 0,Y 250.463,Z 446.874,A -85,B 0,C 180,E1 -18793.704,E2 -18793.704} C_VEL
LIN {X 0,Y 248.439,Z 450.841,A -85,B 0,C 180,E1 -18796.92,E2 -18796.92} C_VEL
LIN {X 0,Y 247.867,Z 452.257,A -85,B 0,C 180,E1 -18798.552,E2 -18798.552} C_VEL
LIN {X 0,Y 247.339,Z 453.914,A -85,B 0,C 180,E1 -18801.832,E2 -18801.832} C_VEL
LIN {X 0,Y 247.437,Z 454.203,A -85,B 0,C 180,E1 -18803.794,E2 -18803.794} C_VEL
LIN {X 0,Y 247.863,Z 453.525,A -85,B 0,C 180,E1 -18806.749,E2 -18806.749} C_VEL
LIN {X 0,Y 248.201,Z 452.586,A -85,B 0,C 180,E1 -18808.377,E2 -18808.377} C_VEL
LIN {X 0,Y 248.596,Z 449.751,A -85,B 0,C 180,E1 -18811.215,E2 -18811.215} C_VEL
LIN {X 0,Y 248.493,Z 449.93,A -85,B 0,C 180,E1 -18811.621,E2 -18811.621} C_VEL
LIN {X 0,Y 248.021,Z 451.522,A -85,B 0,C 180,E1 -18813.249,E2 -18813.249} C_VEL
LIN {X 0,Y 247.676,Z 452.454,A -85,B 0,C 180,E1 -18814.883,E2 -18814.883} C_VEL
LIN {X 0,Y 247.543,Z 452.777,A -85,B 0,C 180,E1 -18816.521,E2 -18816.521} C_VEL
LIN {X 0,Y 247.569,Z 452.489,A -85,B 0,C 180,E1 -18818.16,E2 -18818.16} C_VEL
LIN {X 0,Y 247.809,Z 451.599,A -85,B 0,C 180,E1 -18819.797,E2 -18819.797} C_VEL
LIN {X 0,Y 248.613,Z 449.117,A -85,B 0,C 180,E1 -18822.241,E2 -18822.241} C_VEL
LIN {X 0,Y 250.045,Z 445.251,A -85,B 0,C 180,E1 -18824.653,E2 -18824.653} C_VEL
LIN {X 0,Y 252.157,Z 439.822,A -85,B 0,C 180,E1 -18827.017,E2 -18827.017} C_VEL
LIN {X 0,Y 254.726,Z 432.48,A -85,B 0,C 180,E1 -18829.335,E2 -18829.335} C_VEL
LIN {X 0,Y 257.411,Z 424.56,A -85,B 0,C 180,E1 -18831.208,E2 -18831.208} C_VEL
LIN {X 0,Y 259.679,Z 417.105,A -85,B 0,C 180,E1 -18832.586,E2 -18832.586} C_VEL
LIN {X 0,Y 261.802,Z 409.308,A -85,B 0,C 180,E1 -18833.745,E2 -18833.745} C_VEL
LIN {X 0,Y 262.796,Z 399.781,A -85,B 0,C 180,E1 -18835.122,E2 -18835.122} C_VEL
LIN {X 0,Y 263.296,Z 392.264,A -85,B 0,C 180,E1 -18836.05,E2 -18836.05} C_VEL
LIN {X 0,Y 261.915,Z 381.71,A -85,B 0,C 180,E1 -18837.685,E2 -18837.685} C_VEL
LIN {X 0,Y 263.113,Z 373.261,A -85,B 0,C 180,E1 -18840.035,E2 -18840.035} C_VEL
LIN {X 0,Y 265.316,Z 363.195,A -85,B 0,C 180,E1 -18843.343,E2 -18843.343} C_VEL
LIN {X 0,Y 265.379,Z 360.288,A -85,B 0,C 180,E1 -18844.816,E2 -18844.816} C_VEL
LIN {X 0,Y 265.169,Z 356.234,A -85,B 0,C 180,E1 -18847.56,E2 -18847.56} C_VEL
LIN {X 0,Y 265.019,Z 353.95,A -85,B 0,C 180,E1 -18849.729,E2 -18849.729} C_VEL
LIN {X 0,Y 264.557,Z 352.588,A -85,B 0,C 180,E1 -18851.94,E2 -18851.94} C_VEL
LIN {X 0,Y 263.973,Z 352.014,A -85,B 0,C 180,E1 -18854.038,E2 -18854.038} C_VEL
LIN {X 0,Y 263.467,Z 351.914,A -85,B 0,C 180,E1 -18856.086,E2 -18856.086} C_VEL
LIN {X 0,Y 262.993,Z 352.266,A -85,B 0,C 180,E1 -18858.439,E2 -18858.439} C_VEL
LIN {X 0,Y 262.489,Z 353.612,A -85,B 0,C 180,E1 -18861.987,E2 -18861.987} C_VEL
LIN {X 0,Y 262.272,Z 354.691,A -85,B 0,C 180,E1 -18863.875,E2 -18863.875} C_VEL
LIN {X 0,Y 261.911,Z 356.504,A -85,B 0,C 180,E1 -18866.289,E2 -18866.289} C_VEL
LIN {X 0,Y 261.598,Z 357.622,A -85,B 0,C 180,E1 -18867.497,E2 -18867.497} C_VEL
LIN {X 0,Y 260.721,Z 359.974,A -85,B 0,C 180,E1 -18869.61,E2 -18869.61} C_VEL
LIN {X 0,Y 259.775,Z 362.874,A -85,B 0,C 180,E1 -18871.801,E2 -18871.801} C_VEL
LIN {X 0,Y 263.281,Z 373.027,A -85,B 0,C 180,E1 -18874.714,E2 -18874.714} C_VEL
LIN {X 0,Y 265.095,Z 381.529,A -85,B 0,C 180,E1 -18877.035,E2 -18877.035} C_VEL
LIN {X 0,Y 265.716,Z 388.78,A -85,B 0,C 180,E1 -18879.077,E2 -18879.077} C_VEL
LIN {X 0,Y 265.622,Z 391.577,A -85,B 0,C 180,E1 -18879.88,E2 -18879.88} C_VEL
LIN {X 0,Y 263.324,Z 397.417,A -85,B 0,C 180,E1 -18881.319,E2 -18881.319} C_VEL
LIN {X 0,Y 260.988,Z 402.201,A -85,B 0,C 180,E1 -18882.768,E2 -18882.768} C_VEL
LIN {X 0,Y 257.907,Z 407.546,A -85,B 0,C 180,E1 -18884.995,E2 -18884.995} C_VEL
LIN {X 0,Y 256.109,Z 410.089,A -85,B 0,C 180,E1 -18886.509,E2 -18886.509} C_VEL
LIN {X 0,Y 253.644,Z 412.505,A -85,B 0,C 180,E1 -18888.814,E2 -18888.814} C_VEL
LIN {X 0,Y 252.123,Z 413.333,A -85,B 0,C 180,E1 -18890.37,E2 -18890.37} C_VEL
LIN {X 0,Y 250.77,Z 413.516,A -85,B 0,C 180,E1 -18891.943,E2 -18891.943} C_VEL
LIN {X 0,Y 249.699,Z 413.024,A -85,B 0,C 180,E1 -18893.534,E2 -18893.534} C_VEL
LIN {X 0,Y 248.857,Z 411.874,A -85,B 0,C 180,E1 -18895.138,E2 -18895.138} C_VEL
LIN {X 0,Y 248.027,Z 408.866,A -85,B 0,C 180,E1 -18897.562,E2 -18897.562} C_VEL
LIN {X 0,Y 247.702,Z 405.976,A -85,B 0,C 180,E1 -18899.185,E2 -18899.185} C_VEL
LIN {X 0,Y 247.501,Z 401.252,A -85,B 0,C 180,E1 -18901.218,E2 -18901.218} C_VEL
LIN {X 0,Y 247.617,Z 394.948,A -85,B 0,C 180,E1 -18903.252,E2 -18903.252} C_VEL
LIN {X 0,Y 248.05,Z 386.801,A -85,B 0,C 180,E1 -18905.281,E2 -18905.281} C_VEL
LIN {X 0,Y 248.227,Z 379.255,A -85,B 0,C 180,E1 -18906.754,E2 -18906.754} C_VEL
LIN {X 0,Y 248.528,Z 369.563,A -85,B 0,C 180,E1 -18908.209,E2 -18908.209} C_VEL
LIN {X 0,Y 248.785,Z 359.734,A -85,B 0,C 180,E1 -18909.305,E2 -18909.305} C_VEL
LIN {X 0,Y 248.66,Z 354.433,A -85,B 0,C 180,E1 -18909.761,E2 -18909.761} C_VEL
LIN {X 0,Y 248.46,Z 352.565,A -85,B 0,C 180,E1 -18909.923,E2 -18909.923} C_VEL
LIN {X 0,Y 248.387,Z 341.939,A -85,B 0,C 180,E1 -18915.292,E2 -18915.292} C_VEL
LIN {X 0,Y 248.607,Z 331.852,A -85,B 0,C 180,E1 -18920.48,E2 -18920.48} C_VEL
LIN {X 0,Y 248.891,Z 323.033,A -85,B 0,C 180,E1 -18925.057,E2 -18925.057} C_VEL
LIN {X 0,Y 249.242,Z 314.236,A -85,B 0,C 180,E1 -18929.679,E2 -18929.679} C_VEL
LIN {X 0,Y 249.321,Z 313.426,A -85,B 0,C 180,E1 -18930.179,E2 -18930.179} C_VEL
LIN {X 0,Y 249.059,Z 313.46,A -85,B 0,C 180,E1 -18935.082,E2 -18935.082} C_VEL
LIN {X 0,Y 249.016,Z 313.465,A -85,B 0,C 180,E1 -18938.379,E2 -18938.379} C_VEL
LIN {X 0,Y 248.987,Z 313.469,A -85,B 0,C 180,E1 -18942.787,E2 -18942.787} C_VEL
LIN {X 0,Y 249.002,Z 313.468,A -85,B 0,C 180,E1 -18947.36,E2 -18947.36} C_VEL
LIN {X 0,Y 249.018,Z 313.462,A -85,B 0,C 180,E1 -18951.618,E2 -18951.618} C_VEL
LIN {X 0,Y 249.035,Z 313.462,A -85,B 0,C 180,E1 -18955.638,E2 -18955.638} C_VEL
LIN {X 0,Y 249.043,Z 313.459,A -85,B 0,C 180,E1 -18959.472,E2 -18959.472} C_VEL
LIN {X 0,Y 249.065,Z 313.459,A -85,B 0,C 180,E1 -18963.161,E2 -18963.161} C_VEL
LIN {X 0,Y 249.072,Z 313.459,A -85,B 0,C 180,E1 -18966.732,E2 -18966.732} C_VEL
LIN {X 0,Y 249.102,Z 313.455,A -85,B 0,C 180,E1 -18970.211,E2 -18970.211} C_VEL
LIN {X 0,Y 249.232,Z 313.438,A -85,B 0,C 180,E1 -18973.621,E2 -18973.621} C_VEL
LIN {X 0,Y 249.224,Z 313.439,A -85,B 0,C 180,E1 -18978.615,E2 -18978.615} C_VEL
LIN {X 0,Y 249.424,Z 313.416,A -85,B 0,C 180,E1 -18981.901,E2 -18981.901} C_VEL
LIN {X 0,Y 249.253,Z 313.433,A -85,B 0,C 180,E1 -18985.148,E2 -18985.148} C_VEL
LIN {X 0,Y 249.646,Z 313.388,A -85,B 0,C 180,E1 -18988.387,E2 -18988.387} C_VEL
LIN {X 0,Y 249.646,Z 313.388,A -85,B 0,C 180,E1 -18991.613,E2 -18991.613} C_VEL
LIN {X 0,Y 249.418,Z 313.414,A -85,B 0,C 180,E1 -18996.472,E2 -18996.472} C_VEL
LIN {X 0,Y 249.332,Z 313.429,A -85,B 0,C 180,E1 -18999.737,E2 -18999.737} C_VEL
LIN {X 0,Y 249.194,Z 313.441,A -85,B 0,C 180,E1 -19004.704,E2 -19004.704} C_VEL
LIN {X 0,Y 249.13,Z 313.451,A -85,B 0,C 180,E1 -19008.078,E2 -19008.078} C_VEL
LIN {X 0,Y 249.094,Z 313.456,A -85,B 0,C 180,E1 -19011.518,E2 -19011.518} C_VEL
LIN {X 0,Y 249.121,Z 313.455,A -85,B 0,C 180,E1 -19015.483,E2 -19015.483} C_VEL
LIN {X 0,Y 249.074,Z 313.458,A -85,B 0,C 180,E1 -19018.995,E2 -19018.995} C_VEL
LIN {X 0,Y 249.022,Z 313.463,A -85,B 0,C 180,E1 -19022.427,E2 -19022.427} C_VEL
LIN {X 0,Y 249.022,Z 313.463,A -85,B 0,C 180,E1 -19026.347,E2 -19026.347} C_VEL
LIN {X 0,Y 248.998,Z 313.466,A -85,B 0,C 180,E1 -19030.48,E2 -19030.48} C_VEL
LIN {X 0,Y 248.978,Z 313.472,A -85,B 0,C 180,E1 -19034.885,E2 -19034.885} C_VEL
LIN {X 0,Y 248.995,Z 313.467,A -85,B 0,C 180,E1 -19037.362,E2 -19037.362} C_VEL
LIN {X 0,Y 249.034,Z 313.463,A -85,B 0,C 180,E1 -19042.203,E2 -19042.203} C_VEL
LIN {X 0,Y 249.328,Z 313.424,A -85,B 0,C 180,E1 -19047.74,E2 -19047.74} C_VEL
LIN {X 0,Y 249.347,Z 313.64,A -85,B 0,C 180,E1 -19048.189,E2 -19048.189} C_VEL
LIN {X 0,Y 249.286,Z 317.201,A -85,B 0,C 180,E1 -19050.923,E2 -19050.923} C_VEL
LIN {X 0,Y 248.649,Z 323.776,A -85,B 0,C 180,E1 -19055.808,E2 -19055.808} C_VEL
LIN {X 0,Y 248.198,Z 329.731,A -85,B 0,C 180,E1 -19060.138,E2 -19060.138} C_VEL
LIN {X 0,Y 247.813,Z 336.044,A -85,B 0,C 180,E1 -19064.633,E2 -19064.633} C_VEL
LIN {X 0,Y 247.698,Z 339.784,A -85,B 0,C 180,E1 -19067.248,E2 -19067.248} C_VEL
LIN {X 0,Y 248.773,Z 352.141,A -85,B 0,C 180,E1 -19068.39,E2 -19068.39} C_VEL
LIN {X 0,Y 249.352,Z 359.488,A -85,B 0,C 180,E1 -19069.24,E2 -19069.24} C_VEL
LIN {X 0,Y 248.822,Z 371.113,A -85,B 0,C 180,E1 -19070.922,E2 -19070.922} C_VEL
LIN {X 0,Y 248.278,Z 380.365,A -85,B 0,C 180,E1 -19072.613,E2 -19072.613} C_VEL
LIN {X 0,Y 248.125,Z 387.975,A -85,B 0,C 180,E1 -19074.313,E2 -19074.313} C_VEL
LIN {X 0,Y 247.674,Z 395.272,A -85,B 0,C 180,E1 -19076.342,E2 -19076.342} C_VEL
LIN {X 0,Y 247.526,Z 401.103,A -85,B 0,C 180,E1 -19078.375,E2 -19078.375} C_VEL
LIN {X 0,Y 247.747,Z 406.549,A -85,B 0,C 180,E1 -19080.815,E2 -19080.815} C_VEL
LIN {X 0,Y 248.283,Z 410.463,A -85,B 0,C 180,E1 -19083.247,E2 -19083.247} C_VEL
LIN {X 0,Y 248.874,Z 412.302,A -85,B 0,C 180,E1 -19084.862,E2 -19084.862} C_VEL
LIN {X 0,Y 249.695,Z 413.552,A -85,B 0,C 180,E1 -19086.466,E2 -19086.466} C_VEL
LIN {X 0,Y 250.727,Z 414.206,A -85,B 0,C 180,E1 -19088.059,E2 -19088.059} C_VEL
LIN {X 0,Y 251.995,Z 414.297,A -85,B 0,C 180,E1 -19089.635,E2 -19089.635} C_VEL
LIN {X 0,Y 253.587,Z 413.829,A -85,B 0,C 180,E1 -19091.188,E2 -19091.188} C_VEL
LIN {X 0,Y 255.225,Z 412.802,A -85,B 0,C 180,E1 -19092.728,E2 -19092.728} C_VEL
LIN {X 0,Y 258.092,Z 410.186,A -85,B 0,C 180,E1 -19094.994,E2 -19094.994} C_VEL
LIN {X 0,Y 261.354,Z 406.32,A -85,B 0,C 180,E1 -19097.207,E2 -19097.207} C_VEL
LIN {X 0,Y 265.075,Z 400.966,A -85,B 0,C 180,E1 -19099.357,E2 -19099.357} C_VEL
LIN {X 0,Y 268.384,Z 395.315,A -85,B 0,C 180,E1 -19101.106,E2 -19101.106} C_VEL
LIN {X 0,Y 269.276,Z 390.033,A -85,B 0,C 180,E1 -19103.049,E2 -19103.049} C_VEL
LIN {X 0,Y 269.459,Z 383.17,A -85,B 0,C 180,E1 -19105.609,E2 -19105.609} C_VEL
LIN {X 0,Y 268.997,Z 376.926,A -85,B 0,C 180,E1 -19108.054,E2 -19108.054} C_VEL
LIN {X 0,Y 267.945,Z 370.18,A -85,B 0,C 180,E1 -19111.049,E2 -19111.049} C_VEL
LIN {X 0,Y 266.609,Z 365.999,A -85,B 0,C 180,E1 -19113.615,E2 -19113.615} C_VEL
LIN {X 0,Y 265.775,Z 363.51,A -85,B 0,C 180,E1 -19115.576,E2 -19115.576} C_VEL
LIN {X 0,Y 264.561,Z 361.868,A -85,B 0,C 180,E1 -19118.458,E2 -19118.458} C_VEL
LIN {X 0,Y 264.217,Z 361.872,A -85,B 0,C 180,E1 -19119.307,E2 -19119.307} C_VEL
LIN {X 0,Y 263.459,Z 362.876,A -85,B 0,C 180,E1 -19120.565,E2 -19120.565} C_VEL
LIN {X 0,Y 261.591,Z 368.398,A -85,B 0,C 180,E1 -19124.295,E2 -19124.295} C_VEL
LIN {X 0,Y 261.701,Z 369.214,A -85,B 0,C 180,E1 -19125.156,E2 -19125.156} C_VEL
LIN {X 0,Y 263.211,Z 372.247,A -85,B 0,C 180,E1 -19128.388,E2 -19128.388} C_VEL
LIN {X 0,Y 263.928,Z 373.384,A -85,B 0,C 180,E1 -19129.353,E2 -19129.353} C_VEL
LIN {X 0,Y 266.384,Z 379.405,A -85,B 0,C 180,E1 -19132.641,E2 -19132.641} C_VEL
LIN {X 0,Y 267.317,Z 382.482,A -85,B 0,C 180,E1 -19133.895,E2 -19133.895} C_VEL
LIN {X 0,Y 267.196,Z 387.173,A -85,B 0,C 180,E1 -19135.09,E2 -19135.09} C_VEL
LIN {X 0,Y 265.924,Z 398.658,A -85,B 0,C 180,E1 -19137.751,E2 -19137.751} C_VEL
LIN {X 0,Y 264.169,Z 407.003,A -85,B 0,C 180,E1 -19139.637,E2 -19139.637} C_VEL
LIN {X 0,Y 262,Z 413.613,A -85,B 0,C 180,E1 -19141.129,E2 -19141.129} C_VEL
LIN {X 0,Y 257.584,Z 422.672,A -85,B 0,C 180,E1 -19143.244,E2 -19143.244} C_VEL
LIN {X 0,Y 253.38,Z 430.215,A -85,B 0,C 180,E1 -19145.414,E2 -19145.414} C_VEL
LIN {X 0,Y 249.754,Z 436.469,A -85,B 0,C 180,E1 -19147.673,E2 -19147.673} C_VEL
LIN {X 0,Y 246.502,Z 441.932,A -85,B 0,C 180,E1 -19150.201,E2 -19150.201} C_VEL
LIN {X 0,Y 243.629,Z 446.817,A -85,B 0,C 180,E1 -19153.233,E2 -19153.233} C_VEL
LIN {X 0,Y 242.524,Z 448.852,A -85,B 0,C 180,E1 -19154.882,E2 -19154.882} C_VEL
LIN {X 0,Y 241.506,Z 450.463,A -85,B 0,C 180,E1 -19156.538,E2 -19156.538} C_VEL
LIN {X 0,Y 240.498,Z 452.62,A -85,B 0,C 180,E1 -19159.902,E2 -19159.902} C_VEL
LIN {X 0,Y 240.32,Z 453.252,A -85,B 0,C 180,E1 -19163.282,E2 -19163.282} C_VEL
LIN {X 0,Y 240.83,Z 452.375,A -85,B 0,C 180,E1 -19166.654,E2 -19166.654} C_VEL
LIN {X 0,Y 241.223,Z 451.281,A -85,B 0,C 180,E1 -19168.33,E2 -19168.33} C_VEL
LIN {X 0,Y 241.642,Z 448.766,A -85,B 0,C 180,E1 -19170.833,E2 -19170.833} C_VEL
LIN {X 0,Y 241.639,Z 448.099,A -85,B 0,C 180,E1 -19171.458,E2 -19171.458} C_VEL
LIN {X 0,Y 241.027,Z 450.197,A -85,B 0,C 180,E1 -19173.343,E2 -19173.343} C_VEL
LIN {X 0,Y 240.654,Z 451.339,A -85,B 0,C 180,E1 -19175.026,E2 -19175.026} C_VEL
LIN {X 0,Y 240.507,Z 451.85,A -85,B 0,C 180,E1 -19176.712,E2 -19176.712} C_VEL
LIN {X 0,Y 240.545,Z 451.762,A -85,B 0,C 180,E1 -19178.4,E2 -19178.4} C_VEL
LIN {X 0,Y 240.773,Z 451.079,A -85,B 0,C 180,E1 -19180.087,E2 -19180.087} C_VEL
LIN {X 0,Y 241.285,Z 449.815,A -85,B 0,C 180,E1 -19181.765,E2 -19181.765} C_VEL
LIN {X 0,Y 242.625,Z 446.806,A -85,B 0,C 180,E1 -19184.254,E2 -19184.254} C_VEL
LIN {X 0,Y 244.594,Z 442.372,A -85,B 0,C 180,E1 -19186.698,E2 -19186.698} C_VEL
LIN {X 0,Y 246.761,Z 437.411,A -85,B 0,C 180,E1 -19188.688,E2 -19188.688} C_VEL
LIN {X 0,Y 249.263,Z 431.12,A -85,B 0,C 180,E1 -19190.637,E2 -19190.637} C_VEL
LIN {X 0,Y 252.224,Z 423.168,A -85,B 0,C 180,E1 -19192.528,E2 -19192.528} C_VEL
LIN {X 0,Y 255.063,Z 415.052,A -85,B 0,C 180,E1 -19194.004,E2 -19194.004} C_VEL
LIN {X 0,Y 256.652,Z 408.663,A -85,B 0,C 180,E1 -19195.008,E2 -19195.008} C_VEL
LIN {X 0,Y 258.027,Z 398.413,A -85,B 0,C 180,E1 -19196.54,E2 -19196.54} C_VEL
LIN {X 0,Y 258.256,Z 393.5,A -85,B 0,C 180,E1 -19197.222,E2 -19197.222} C_VEL
LIN {X 0,Y 257.044,Z 383.078,A -85,B 0,C 180,E1 -19199.007,E2 -19199.007} C_VEL
LIN {X 0,Y 256.793,Z 380.447,A -85,B 0,C 180,E1 -19199.514,E2 -19199.514} C_VEL
LIN {X 0,Y 258.47,Z 371.666,A -85,B 0,C 180,E1 -19202.247,E2 -19202.247} C_VEL
LIN {X 0,Y 259.639,Z 367.42,A -85,B 0,C 180,E1 -19203.704,E2 -19203.704} C_VEL
LIN {X 0,Y 259.856,Z 365.452,A -85,B 0,C 180,E1 -19204.608,E2 -19204.608} C_VEL
LIN {X 0,Y 259.721,Z 362.3,A -85,B 0,C 180,E1 -19206.535,E2 -19206.535} C_VEL
LIN {X 0,Y 259.618,Z 359.74,A -85,B 0,C 180,E1 -19208.508,E2 -19208.508} C_VEL
LIN {X 0,Y 259.3,Z 357.807,A -85,B 0,C 180,E1 -19210.63,E2 -19210.63} C_VEL
LIN {X 0,Y 258.707,Z 356.713,A -85,B 0,C 180,E1 -19212.819,E2 -19212.819} C_VEL
LIN {X 0,Y 258.027,Z 356.273,A -85,B 0,C 180,E1 -19215.087,E2 -19215.087} C_VEL
LIN {X 0,Y 257.422,Z 356.323,A -85,B 0,C 180,E1 -19217.489,E2 -19217.489} C_VEL
LIN {X 0,Y 256.776,Z 357.21,A -85,B 0,C 180,E1 -19220.984,E2 -19220.984} C_VEL
LIN {X 0,Y 256.457,Z 358.118,A -85,B 0,C 180,E1 -19222.921,E2 -19222.921} C_VEL
LIN {X 0,Y 256.046,Z 359.71,A -85,B 0,C 180,E1 -19225.432,E2 -19225.432} C_VEL
LIN {X 0,Y 255.746,Z 360.688,A -85,B 0,C 180,E1 -19226.658,E2 -19226.658} C_VEL
LIN {X 0,Y 254.62,Z 363.482,A -85,B 0,C 180,E1 -19229.386,E2 -19229.386} C_VEL
LIN {X 0,Y 254.43,Z 364.113,A -85,B 0,C 180,E1 -19229.824,E2 -19229.824} C_VEL
LIN {X 0,Y 257.358,Z 373.043,A -85,B 0,C 180,E1 -19232.708,E2 -19232.708} C_VEL
LIN {X 0,Y 258.923,Z 379.718,A -85,B 0,C 180,E1 -19234.756,E2 -19234.756} C_VEL
LIN {X 0,Y 259.847,Z 386.735,A -85,B 0,C 180,E1 -19236.866,E2 -19236.866} C_VEL
LIN {X 0,Y 259.84,Z 393.333,A -85,B 0,C 180,E1 -19238.942,E2 -19238.942} C_VEL
LIN {X 0,Y 259.527,Z 394.917,A -85,B 0,C 180,E1 -19239.386,E2 -19239.386} C_VEL
LIN {X 0,Y 256.297,Z 401.512,A -85,B 0,C 180,E1 -19241.202,E2 -19241.202} C_VEL
LIN {X 0,Y 253.412,Z 406.501,A -85,B 0,C 180,E1 -19243.068,E2 -19243.068} C_VEL
LIN {X 0,Y 250.325,Z 410.676,A -85,B 0,C 180,E1 -19245.362,E2 -19245.362} C_VEL
LIN {X 0,Y 248.484,Z 412.598,A -85,B 0,C 180,E1 -19246.921,E2 -19246.921} C_VEL
LIN {X 0,Y 246.814,Z 413.821,A -85,B 0,C 180,E1 -19248.501,E2 -19248.501} C_VEL
LIN {X 0,Y 245.2,Z 414.402,A -85,B 0,C 180,E1 -19250.095,E2 -19250.095} C_VEL
LIN {X 0,Y 243.795,Z 414.327,A -85,B 0,C 180,E1 -19251.711,E2 -19251.711} C_VEL
LIN {X 0,Y 242.677,Z 413.592,A -85,B 0,C 180,E1 -19253.346,E2 -19253.346} C_VEL
LIN {X 0,Y 241.452,Z 411.216,A -85,B 0,C 180,E1 -19255.825,E2 -19255.825} C_VEL
LIN {X 0,Y 240.723,Z 407.319,A -85,B 0,C 180,E1 -19258.325,E2 -19258.325} C_VEL
LIN {X 0,Y 240.453,Z 402.772,A -85,B 0,C 180,E1 -19260.416,E2 -19260.416} C_VEL
LIN {X 0,Y 240.469,Z 396.781,A -85,B 0,C 180,E1 -19262.51,E2 -19262.51} C_VEL
LIN {X 0,Y 240.724,Z 390.697,A -85,B 0,C 180,E1 -19264.183,E2 -19264.183} C_VEL
LIN {X 0,Y 241.119,Z 383.092,A -85,B 0,C 180,E1 -19265.853,E2 -19265.853} C_VEL
LIN {X 0,Y 241.268,Z 374.6,A -85,B 0,C 180,E1 -19267.326,E2 -19267.326} C_VEL
LIN {X 0,Y 241.555,Z 365.16,A -85,B 0,C 180,E1 -19268.573,E2 -19268.573} C_VEL
LIN {X 0,Y 241.729,Z 355.695,A -85,B 0,C 180,E1 -19269.516,E2 -19269.516} C_VEL
LIN {X 0,Y 241.423,Z 353.213,A -85,B 0,C 180,E1 -19269.739,E2 -19269.739} C_VEL
LIN {X 0,Y 241.303,Z 342.562,A -85,B 0,C 180,E1 -19275.194,E2 -19275.194} C_VEL
LIN {X 0,Y 241.533,Z 332.507,A -85,B 0,C 180,E1 -19280.434,E2 -19280.434} C_VEL
LIN {X 0,Y 241.804,Z 324.077,A -85,B 0,C 180,E1 -19284.88,E2 -19284.88} C_VEL
LIN {X 0,Y 242.158,Z 315.426,A -85,B 0,C 180,E1 -19289.463,E2 -19289.463} C_VEL
LIN {X 0,Y 242.253,Z 314.307,A -85,B 0,C 180,E1 -19290.146,E2 -19290.146} C_VEL
LIN {X 0,Y 242.001,Z 314.339,A -85,B 0,C 180,E1 -19295.594,E2 -19295.594} C_VEL
LIN {X 0,Y 241.936,Z 314.347,A -85,B 0,C 180,E1 -19299.72,E2 -19299.72} C_VEL
LIN {X 0,Y 241.909,Z 314.348,A -85,B 0,C 180,E1 -19304.203,E2 -19304.203} C_VEL
LIN {X 0,Y 241.926,Z 314.348,A -85,B 0,C 180,E1 -19308.075,E2 -19308.075} C_VEL
LIN {X 0,Y 241.979,Z 314.34,A -85,B 0,C 180,E1 -19312.416,E2 -19312.416} C_VEL
LIN {X 0,Y 241.972,Z 314.344,A -85,B 0,C 180,E1 -19316.506,E2 -19316.506} C_VEL
LIN {X 0,Y 242.028,Z 314.336,A -85,B 0,C 180,E1 -19320.586,E2 -19320.586} C_VEL
LIN {X 0,Y 242.058,Z 314.333,A -85,B 0,C 180,E1 -19324.182,E2 -19324.182} C_VEL
LIN {X 0,Y 242.044,Z 314.334,A -85,B 0,C 180,E1 -19328.296,E2 -19328.296} C_VEL
LIN {X 0,Y 242.153,Z 314.319,A -85,B 0,C 180,E1 -19333.277,E2 -19333.277} C_VEL
LIN {X 0,Y 242.139,Z 314.32,A -85,B 0,C 180,E1 -19336.573,E2 -19336.573} C_VEL
LIN {X 0,Y 242.374,Z 314.293,A -85,B 0,C 180,E1 -19341.664,E2 -19341.664} C_VEL
LIN {X 0,Y 242.215,Z 314.309,A -85,B 0,C 180,E1 -19345.006,E2 -19345.006} C_VEL
LIN {X 0,Y 242.606,Z 314.265,A -85,B 0,C 180,E1 -19348.34,E2 -19348.34} C_VEL
LIN {X 0,Y 242.606,Z 314.265,A -85,B 0,C 180,E1 -19351.66,E2 -19351.66} C_VEL
LIN {X 0,Y 242.39,Z 314.289,A -85,B 0,C 180,E1 -19356.66,E2 -19356.66} C_VEL
LIN {X 0,Y 242.255,Z 314.308,A -85,B 0,C 180,E1 -19360.024,E2 -19360.024} C_VEL
LIN {X 0,Y 242.156,Z 314.319,A -85,B 0,C 180,E1 -19365.142,E2 -19365.142} C_VEL
LIN {X 0,Y 242.069,Z 314.329,A -85,B 0,C 180,E1 -19368.624,E2 -19368.624} C_VEL
LIN {X 0,Y 242.04,Z 314.332,A -85,B 0,C 180,E1 -19372.177,E2 -19372.177} C_VEL
LIN {X 0,Y 242.057,Z 314.333,A -85,B 0,C 180,E1 -19375.839,E2 -19375.839} C_VEL
LIN {X 0,Y 242.021,Z 314.336,A -85,B 0,C 180,E1 -19379.581,E2 -19379.581} C_VEL
LIN {X 0,Y 241.972,Z 314.344,A -85,B 0,C 180,E1 -19383.494,E2 -19383.494} C_VEL
LIN {X 0,Y 241.979,Z 314.34,A -85,B 0,C 180,E1 -19387.584,E2 -19387.584} C_VEL
LIN {X 0,Y 241.926,Z 314.348,A -85,B 0,C 180,E1 -19391.925,E2 -19391.925} C_VEL
LIN {X 0,Y 241.914,Z 314.349,A -85,B 0,C 180,E1 -19396.577,E2 -19396.577} C_VEL
LIN {X 0,Y 241.986,Z 314.34,A -85,B 0,C 180,E1 -19401.643,E2 -19401.643} C_VEL
LIN {X 0,Y 242.125,Z 314.323,A -85,B 0,C 180,E1 -19406.533,E2 -19406.533} C_VEL
LIN {X 0,Y 242.298,Z 314.407,A -85,B 0,C 180,E1 -19408.11,E2 -19408.11} C_VEL
LIN {X 0,Y 242.254,Z 317.438,A -85,B 0,C 180,E1 -19410.497,E2 -19410.497} C_VEL
LIN {X 0,Y 241.746,Z 322.45,A -85,B 0,C 180,E1 -19414.321,E2 -19414.321} C_VEL
LIN {X 0,Y 241.286,Z 328.389,A -85,B 0,C 180,E1 -19418.761,E2 -19418.761} C_VEL
LIN {X 0,Y 240.852,Z 334.23,A -85,B 0,C 180,E1 -19423.037,E2 -19423.037} C_VEL
LIN {X 0,Y 240.621,Z 340.083,A -85,B 0,C 180,E1 -19427.241,E2 -19427.241} C_VEL
LIN {X 0,Y 241.712,Z 352.805,A -85,B 0,C 180,E1 -19428.471,E2 -19428.471} C_VEL
LIN {X 0,Y 242.208,Z 360.085,A -85,B 0,C 180,E1 -19429.342,E2 -19429.342} C_VEL
LIN {X 0,Y 241.708,Z 371.338,A -85,B 0,C 180,E1 -19431.011,E2 -19431.011} C_VEL
LIN {X 0,Y 241.175,Z 381.604,A -85,B 0,C 180,E1 -19432.967,E2 -19432.967} C_VEL
LIN {X 0,Y 240.98,Z 388.441,A -85,B 0,C 180,E1 -19434.563,E2 -19434.563} C_VEL
LIN {X 0,Y 240.55,Z 395.774,A -85,B 0,C 180,E1 -19436.652,E2 -19436.652} C_VEL
LIN {X 0,Y 240.471,Z 402.724,A -85,B 0,C 180,E1 -19439.165,E2 -19439.165} C_VEL
LIN {X 0,Y 240.736,Z 407.933,A -85,B 0,C 180,E1 -19441.675,E2 -19441.675} C_VEL
LIN {X 0,Y 241.505,Z 411.656,A -85,B 0,C 180,E1 -19444.174,E2 -19444.174} C_VEL
LIN {X 0,Y 242.674,Z 414.058,A -85,B 0,C 180,E1 -19446.654,E2 -19446.654} C_VEL
LIN {X 0,Y 243.756,Z 414.947,A -85,B 0,C 180,E1 -19448.291,E2 -19448.291} C_VEL
LIN {X 0,Y 245.059,Z 415.243,A -85,B 0,C 180,E1 -19449.91,E2 -19449.91} C_VEL
LIN {X 0,Y 246.731,Z 414.97,A -85,B 0,C 180,E1 -19451.503,E2 -19451.503} C_VEL
LIN {X 0,Y 248.428,Z 414.186,A -85,B 0,C 180,E1 -19453.082,E2 -19453.082} C_VEL
LIN {X 0,Y 250.401,Z 412.835,A -85,B 0,C 180,E1 -19454.634,E2 -19454.634} C_VEL
LIN {X 0,Y 253.656,Z 409.768,A -85,B 0,C 180,E1 -19456.915,E2 -19456.915} C_VEL
LIN {X 0,Y 257.385,Z 405.351,A -85,B 0,C 180,E1 -19459.129,E2 -19459.129} C_VEL
LIN {X 0,Y 261.485,Z 399.548,A -85,B 0,C 180,E1 -19461.277,E2 -19461.277} C_VEL
LIN {X 0,Y 262.723,Z 397.346,A -85,B 0,C 180,E1 -19461.996,E2 -19461.996} C_VEL
LIN {X 0,Y 263.923,Z 390.804,A -85,B 0,C 180,E1 -19464.643,E2 -19464.643} C_VEL
LIN {X 0,Y 264.203,Z 383.343,A -85,B 0,C 180,E1 -19467.746,E2 -19467.746} C_VEL
LIN {X 0,Y 263.686,Z 376.402,A -85,B 0,C 180,E1 -19471.016,E2 -19471.016} C_VEL
LIN {X 0,Y 263.093,Z 372.873,A -85,B 0,C 180,E1 -19473.107,E2 -19473.107} C_VEL
LIN {X 0,Y 262.06,Z 369.345,A -85,B 0,C 180,E1 -19476.159,E2 -19476.159} C_VEL
LIN {X 0,Y 261.245,Z 368.077,A -85,B 0,C 180,E1 -19478.725,E2 -19478.725} C_VEL
LIN {X 0,Y 261.043,Z 367.665,A -85,B 0,C 180,E1 -19481.076,E2 -19481.076} C_VEL
LIN {X 0,Y 261.265,Z 368.163,A -85,B 0,C 180,E1 -19483.423,E2 -19483.423} C_VEL
LIN {X 0,Y 261.701,Z 369.214,A -85,B 0,C 180,E1 -19485.156,E2 -19485.156} C_VEL
LIN {X 0,Y 261.864,Z 370.793,A -85,B 0,C 180,E1 -19486.402,E2 -19486.402} C_VEL
LIN {X 0,Y 261.678,Z 373.364,A -85,B 0,C 180,E1 -19487.578,E2 -19487.578} C_VEL
LIN {X 0,Y 261.137,Z 381.604,A -85,B 0,C 180,E1 -19490.61,E2 -19490.61} C_VEL
LIN {X 0,Y 261.498,Z 383.281,A -85,B 0,C 180,E1 -19491.408,E2 -19491.408} C_VEL
LIN {X 0,Y 262.349,Z 385.532,A -85,B 0,C 180,E1 -19492.591,E2 -19492.591} C_VEL
LIN {X 0,Y 262.717,Z 387.975,A -85,B 0,C 180,E1 -19493.536,E2 -19493.536} C_VEL
LIN {X 0,Y 261.275,Z 397.99,A -85,B 0,C 180,E1 -19496.072,E2 -19496.072} C_VEL
LIN {X 0,Y 259.078,Z 407.406,A -85,B 0,C 180,E1 -19498.381,E2 -19498.381} C_VEL
LIN {X 0,Y 256.046,Z 415.685,A -85,B 0,C 180,E1 -19500.392,E2 -19500.392} C_VEL
LIN {X 0,Y 251.371,Z 424.191,A -85,B 0,C 180,E1 -19502.528,E2 -19502.528} C_VEL
LIN {X 0,Y 247.026,Z 431.243,A -85,B 0,C 180,E1 -19504.738,E2 -19504.738} C_VEL
LIN {X 0,Y 243.226,Z 437.086,A -85,B 0,C 180,E1 -19507.04,E2 -19507.04} C_VEL
LIN {X 0,Y 239.635,Z 442.516,A -85,B 0,C 180,E1 -19509.805,E2 -19509.805} C_VEL
LIN {X 0,Y 236.82,Z 446.733,A -85,B 0,C 180,E1 -19512.737,E2 -19512.737} C_VEL
LIN {X 0,Y 234.59,Z 450.057,A -85,B 0,C 180,E1 -19516.133,E2 -19516.133} C_VEL
LIN {X 0,Y 233.496,Z 451.891,A -85,B 0,C 180,E1 -19519.596,E2 -19519.596} C_VEL
LIN {X 0,Y 233.285,Z 452.28,A -85,B 0,C 180,E1 -19523.079,E2 -19523.079} C_VEL
LIN {X 0,Y 233.499,Z 451.893,A -85,B 0,C 180,E1 -19524.819,E2 -19524.819} C_VEL
LIN {X 0,Y 233.822,Z 451.106,A -85,B 0,C 180,E1 -19526.554,E2 -19526.554} C_VEL
LIN {X 0,Y 234.254,Z 449.92,A -85,B 0,C 180,E1 -19528.281,E2 -19528.281} C_VEL
LIN {X 0,Y 234.7,Z 447.211,A -85,B 0,C 180,E1 -19530.858,E2 -19530.858} C_VEL
LIN {X 0,Y 234.738,Z 446.437,A -85,B 0,C 180,E1 -19531.501,E2 -19531.501} C_VEL
LIN {X 0,Y 234.085,Z 448.729,A -85,B 0,C 180,E1 -19533.443,E2 -19533.443} C_VEL
LIN {X 0,Y 233.672,Z 450.054,A -85,B 0,C 180,E1 -19535.177,E2 -19535.177} C_VEL
LIN {X 0,Y 233.484,Z 450.774,A -85,B 0,C 180,E1 -19536.915,E2 -19536.915} C_VEL
LIN {X 0,Y 233.515,Z 450.905,A -85,B 0,C 180,E1 -19538.655,E2 -19538.655} C_VEL
LIN {X 0,Y 233.756,Z 450.453,A -85,B 0,C 180,E1 -19540.393,E2 -19540.393} C_VEL
LIN {X 0,Y 234.321,Z 449.437,A -85,B 0,C 180,E1 -19542.12,E2 -19542.12} C_VEL
LIN {X 0,Y 235.748,Z 446.845,A -85,B 0,C 180,E1 -19544.679,E2 -19544.679} C_VEL
LIN {X 0,Y 237.841,Z 442.827,A -85,B 0,C 180,E1 -19547.187,E2 -19547.187} C_VEL
LIN {X 0,Y 240.614,Z 437.311,A -85,B 0,C 180,E1 -19549.627,E2 -19549.627} C_VEL
LIN {X 0,Y 243.355,Z 431.272,A -85,B 0,C 180,E1 -19551.606,E2 -19551.606} C_VEL
LIN {X 0,Y 246.55,Z 423.695,A -85,B 0,C 180,E1 -19553.521,E2 -19553.521} C_VEL
LIN {X 0,Y 249.54,Z 416.073,A -85,B 0,C 180,E1 -19554.99,E2 -19554.99} C_VEL
LIN {X 0,Y 251.212,Z 410.438,A -85,B 0,C 180,E1 -19555.953,E2 -19555.953} C_VEL
LIN {X 0,Y 252.939,Z 400.813,A -85,B 0,C 180,E1 -19557.511,E2 -19557.511} C_VEL
LIN {X 0,Y 253.431,Z 396.786,A -85,B 0,C 180,E1 -19558.128,E2 -19558.128} C_VEL
LIN {X 0,Y 252.942,Z 388.295,A -85,B 0,C 180,E1 -19559.682,E2 -19559.682} C_VEL
LIN {X 0,Y 251.985,Z 379.513,A -85,B 0,C 180,E1 -19561.413,E2 -19561.413} C_VEL
LIN {X 0,Y 253.722,Z 372.428,A -85,B 0,C 180,E1 -19563.797,E2 -19563.797} C_VEL
LIN {X 0,Y 254.177,Z 370.557,A -85,B 0,C 180,E1 -19564.528,E2 -19564.528} C_VEL
LIN {X 0,Y 254.299,Z 368.723,A -85,B 0,C 180,E1 -19565.477,E2 -19565.477} C_VEL
LIN {X 0,Y 254.195,Z 365.677,A -85,B 0,C 180,E1 -19567.464,E2 -19567.464} C_VEL
LIN {X 0,Y 253.917,Z 363.321,A -85,B 0,C 180,E1 -19569.539,E2 -19569.539} C_VEL
LIN {X 0,Y 253.43,Z 361.715,A -85,B 0,C 180,E1 -19571.725,E2 -19571.725} C_VEL
LIN {X 0,Y 252.721,Z 360.833,A -85,B 0,C 180,E1 -19574.046,E2 -19574.046} C_VEL
LIN {X 0,Y 251.621,Z 360.637,A -85,B 0,C 180,E1 -19577.904,E2 -19577.904} C_VEL
LIN {X 0,Y 251.175,Z 361.012,A -85,B 0,C 180,E1 -19579.941,E2 -19579.941} C_VEL
LIN {X 0,Y 250.762,Z 361.73,A -85,B 0,C 180,E1 -19581.931,E2 -19581.931} C_VEL
LIN {X 0,Y 249.978,Z 363.93,A -85,B 0,C 180,E1 -19585.784,E2 -19585.784} C_VEL
LIN {X 0,Y 249.356,Z 365.552,A -85,B 0,C 180,E1 -19587.56,E2 -19587.56} C_VEL
LIN {X 0,Y 251.199,Z 371.233,A -85,B 0,C 180,E1 -19589.759,E2 -19589.759} C_VEL
LIN {X 0,Y 252.958,Z 378.115,A -85,B 0,C 180,E1 -19592.192,E2 -19592.192} C_VEL
LIN {X 0,Y 254.104,Z 385.411,A -85,B 0,C 180,E1 -19594.632,E2 -19594.632} C_VEL
LIN {X 0,Y 254.392,Z 392.243,A -85,B 0,C 180,E1 -19596.915,E2 -19596.915} C_VEL
LIN {X 0,Y 253.859,Z 397.044,A -85,B 0,C 180,E1 -19598.537,E2 -19598.537} C_VEL
LIN {X 0,Y 250.569,Z 403.115,A -85,B 0,C 180,E1 -19600.329,E2 -19600.329} C_VEL
LIN {X 0,Y 248.084,Z 407.076,A -85,B 0,C 180,E1 -19601.841,E2 -19601.841} C_VEL
LIN {X 0,Y 244.684,Z 411.363,A -85,B 0,C 180,E1 -19604.163,E2 -19604.163} C_VEL
LIN {X 0,Y 241.725,Z 414.021,A -85,B 0,C 180,E1 -19606.548,E2 -19606.548} C_VEL
LIN {X 0,Y 239.957,Z 414.963,A -85,B 0,C 180,E1 -19608.167,E2 -19608.167} C_VEL
LIN {X 0,Y 238.26,Z 415.296,A -85,B 0,C 180,E1 -19609.804,E2 -19609.804} C_VEL
LIN {X 0,Y 236.825,Z 414.968,A -85,B 0,C 180,E1 -19611.465,E2 -19611.465} C_VEL
LIN {X 0,Y 235.66,Z 413.983,A -85,B 0,C 180,E1 -19613.147,E2 -19613.147} C_VEL
LIN {X 0,Y 234.371,Z 411.328,A -85,B 0,C 180,E1 -19615.699,E2 -19615.699} C_VEL
LIN {X 0,Y 233.63,Z 407.015,A -85,B 0,C 180,E1 -19618.274,E2 -19618.274} C_VEL
LIN {X 0,Y 233.371,Z 402.08,A -85,B 0,C 180,E1 -19620.429,E2 -19620.429} C_VEL
LIN {X 0,Y 233.441,Z 395.668,A -85,B 0,C 180,E1 -19622.586,E2 -19622.586} C_VEL
LIN {X 0,Y 233.716,Z 389.186,A -85,B 0,C 180,E1 -19624.309,E2 -19624.309} C_VEL
LIN {X 0,Y 234.074,Z 382.217,A -85,B 0,C 180,E1 -19625.814,E2 -19625.814} C_VEL
LIN {X 0,Y 234.238,Z 373.386,A -85,B 0,C 180,E1 -19627.307,E2 -19627.307} C_VEL
LIN {X 0,Y 234.547,Z 363.258,A -85,B 0,C 180,E1 -19628.614,E2 -19628.614} C_VEL
LIN {X 0,Y 234.597,Z 355.197,A -85,B 0,C 180,E1 -19629.373,E2 -19629.373} C_VEL
LIN {X 0,Y 234.432,Z 353.935,A -85,B 0,C 180,E1 -19629.488,E2 -19629.488} C_VEL
LIN {X 0,Y 234.233,Z 342.062,A -85,B 0,C 180,E1 -19635.664,E2 -19635.664} C_VEL
LIN {X 0,Y 234.486,Z 331.845,A -85,B 0,C 180,E1 -19641.077,E2 -19641.077} C_VEL
LIN {X 0,Y 234.849,Z 322.413,A -85,B 0,C 180,E1 -19646.133,E2 -19646.133} C_VEL
LIN {X 0,Y 235.192,Z 315.187,A -85,B 0,C 180,E1 -19650.141,E2 -19650.141} C_VEL
LIN {X 0,Y 234.942,Z 315.215,A -85,B 0,C 180,E1 -19654.633,E2 -19654.633} C_VEL
LIN {X 0,Y 234.906,Z 315.225,A -85,B 0,C 180,E1 -19658.933,E2 -19658.933} C_VEL
LIN {X 0,Y 234.867,Z 315.226,A -85,B 0,C 180,E1 -19663.487,E2 -19663.487} C_VEL
LIN {X 0,Y 234.871,Z 315.227,A -85,B 0,C 180,E1 -19666.51,E2 -19666.51} C_VEL
LIN {X 0,Y 234.911,Z 315.221,A -85,B 0,C 180,E1 -19671.077,E2 -19671.077} C_VEL
LIN {X 0,Y 234.919,Z 315.221,A -85,B 0,C 180,E1 -19675.36,E2 -19675.36} C_VEL
LIN {X 0,Y 234.923,Z 315.217,A -85,B 0,C 180,E1 -19679.431,E2 -19679.431} C_VEL
LIN {X 0,Y 234.985,Z 315.212,A -85,B 0,C 180,E1 -19683.792,E2 -19683.792} C_VEL
LIN {X 0,Y 235.002,Z 315.209,A -85,B 0,C 180,E1 -19688.969,E2 -19688.969} C_VEL
LIN {X 0,Y 235.086,Z 315.2,A -85,B 0,C 180,E1 -19693.058,E2 -19693.058} C_VEL
LIN {X 0,Y 235.093,Z 315.198,A -85,B 0,C 180,E1 -19697.921,E2 -19697.921} C_VEL
LIN {X 0,Y 235.308,Z 315.172,A -85,B 0,C 180,E1 -19701.411,E2 -19701.411} C_VEL
LIN {X 0,Y 235.342,Z 315.167,A -85,B 0,C 180,E1 -19703.14,E2 -19703.14} C_VEL
LIN {X 0,Y 235.565,Z 315.142,A -85,B 0,C 180,E1 -19708.29,E2 -19708.29} C_VEL
LIN {X 0,Y 235.565,Z 315.142,A -85,B 0,C 180,E1 -19711.71,E2 -19711.71} C_VEL
LIN {X 0,Y 235.342,Z 315.167,A -85,B 0,C 180,E1 -19716.86,E2 -19716.86} C_VEL
LIN {X 0,Y 235.202,Z 315.185,A -85,B 0,C 180,E1 -19720.328,E2 -19720.328} C_VEL
LIN {X 0,Y 235.103,Z 315.2,A -85,B 0,C 180,E1 -19725.607,E2 -19725.607} C_VEL
LIN {X 0,Y 235.01,Z 315.21,A -85,B 0,C 180,E1 -19729.206,E2 -19729.206} C_VEL
LIN {X 0,Y 234.971,Z 315.213,A -85,B 0,C 180,E1 -19732.882,E2 -19732.882} C_VEL
LIN {X 0,Y 234.961,Z 315.215,A -85,B 0,C 180,E1 -19736.659,E2 -19736.659} C_VEL
LIN {X 0,Y 234.923,Z 315.217,A -85,B 0,C 180,E1 -19740.569,E2 -19740.569} C_VEL
LIN {X 0,Y 234.919,Z 315.221,A -85,B 0,C 180,E1 -19744.64,E2 -19744.64} C_VEL
LIN {X 0,Y 234.934,Z 315.219,A -85,B 0,C 180,E1 -19748.946,E2 -19748.946} C_VEL
LIN {X 0,Y 234.871,Z 315.227,A -85,B 0,C 180,E1 -19753.49,E2 -19753.49} C_VEL
LIN {X 0,Y 234.867,Z 315.226,A -85,B 0,C 180,E1 -19756.513,E2 -19756.513} C_VEL
LIN {X 0,Y 234.912,Z 315.224,A -85,B 0,C 180,E1 -19761.081,E2 -19761.081} C_VEL
LIN {X 0,Y 235.006,Z 315.207,A -85,B 0,C 180,E1 -19765.378,E2 -19765.378} C_VEL
LIN {X 0,Y 235.261,Z 315.258,A -85,B 0,C 180,E1 -19768.107,E2 -19768.107} C_VEL
LIN {X 0,Y 235.245,Z 317.663,A -85,B 0,C 180,E1 -19770.041,E2 -19770.041} C_VEL
LIN {X 0,Y 234.723,Z 322.639,A -85,B 0,C 180,E1 -19773.93,E2 -19773.93} C_VEL
LIN {X 0,Y 234.19,Z 329.121,A -85,B 0,C 180,E1 -19778.895,E2 -19778.895} C_VEL
LIN {X 0,Y 233.731,Z 335.261,A -85,B 0,C 180,E1 -19783.495,E2 -19783.495} C_VEL
LIN {X 0,Y 233.533,Z 340.424,A -85,B 0,C 180,E1 -19787.29,E2 -19787.29} C_VEL
LIN {X 0,Y 234.581,Z 352.303,A -85,B 0,C 180,E1 -19788.445,E2 -19788.445} C_VEL
LIN {X 0,Y 235.143,Z 358.88,A -85,B 0,C 180,E1 -19789.236,E2 -19789.236} C_VEL
LIN {X 0,Y 234.65,Z 370.431,A -85,B 0,C 180,E1 -19790.955,E2 -19790.955} C_VEL
LIN {X 0,Y 234.11,Z 380.508,A -85,B 0,C 180,E1 -19792.865,E2 -19792.865} C_VEL
LIN {X 0,Y 233.838,Z 388.87,A -85,B 0,C 180,E1 -19794.829,E2 -19794.829} C_VEL
LIN {X 0,Y 233.431,Z 396.266,A -85,B 0,C 180,E1 -19796.982,E2 -19796.982} C_VEL
LIN {X 0,Y 233.391,Z 403.211,A -85,B 0,C 180,E1 -19799.571,E2 -19799.571} C_VEL
LIN {X 0,Y 233.644,Z 407.708,A -85,B 0,C 180,E1 -19801.726,E2 -19801.726} C_VEL
LIN {X 0,Y 234.442,Z 411.797,A -85,B 0,C 180,E1 -19804.3,E2 -19804.3} C_VEL
LIN {X 0,Y 235.658,Z 414.48,A -85,B 0,C 180,E1 -19806.853,E2 -19806.853} C_VEL
LIN {X 0,Y 236.771,Z 415.571,A -85,B 0,C 180,E1 -19808.537,E2 -19808.537} C_VEL
LIN {X 0,Y 238.12,Z 416.119,A -85,B 0,C 180,E1 -19810.202,E2 -19810.202} C_VEL
LIN {X 0,Y 239.849,Z 416.063,A -85,B 0,C 180,E1 -19811.838,E2 -19811.838} C_VEL
LIN {X 0,Y 241.635,Z 415.502,A -85,B 0,C 180,E1 -19813.457,E2 -19813.457} C_VEL
LIN {X 0,Y 243.688,Z 414.408,A -85,B 0,C 180,E1 -19815.046,E2 -19815.046} C_VEL
LIN {X 0,Y 247.079,Z 411.705,A -85,B 0,C 180,E1 -19817.379,E2 -19817.379} C_VEL
LIN {X 0,Y 250.979,Z 407.759,A -85,B 0,C 180,E1 -19819.637,E2 -19819.637} C_VEL
LIN {X 0,Y 255.237,Z 402.409,A -85,B 0,C 180,E1 -19821.824,E2 -19821.824} C_VEL
LIN {X 0,Y 256.712,Z 400.328,A -85,B 0,C 180,E1 -19822.539,E2 -19822.539} C_VEL
LIN {X 0,Y 258.076,Z 395.527,A -85,B 0,C 180,E1 -19824.68,E2 -19824.68} C_VEL
LIN {X 0,Y 258.943,Z 389.365,A -85,B 0,C 180,E1 -19827.479,E2 -19827.479} C_VEL
LIN {X 0,Y 259.145,Z 382.984,A -85,B 0,C 180,E1 -19830.634,E2 -19830.634} C_VEL
LIN {X 0,Y 259.156,Z 380.571,A -85,B 0,C 180,E1 -19831.953,E2 -19831.953} C_VEL
LIN {X 0,Y 258.773,Z 377.951,A -85,B 0,C 180,E1 -19833.791,E2 -19833.791} C_VEL
LIN {X 0,Y 258.504,Z 376.236,A -85,B 0,C 180,E1 -19835.351,E2 -19835.351} C_VEL
LIN {X 0,Y 258.154,Z 375.078,A -85,B 0,C 180,E1 -19836.795,E2 -19836.795} C_VEL
LIN {X 0,Y 257.663,Z 373.946,A -85,B 0,C 180,E1 -19840.206,E2 -19840.206} C_VEL
LIN {X 0,Y 257.819,Z 374.282,A -85,B 0,C 180,E1 -19842.962,E2 -19842.962} C_VEL
LIN {X 0,Y 258.281,Z 375.389,A -85,B 0,C 180,E1 -19845.032,E2 -19845.032} C_VEL
LIN {X 0,Y 259.597,Z 378.267,A -85,B 0,C 180,E1 -19848.166,E2 -19848.166} C_VEL
LIN {X 0,Y 260.467,Z 380.166,A -85,B 0,C 180,E1 -19849.641,E2 -19849.641} C_VEL
LIN {X 0,Y 261.498,Z 383.281,A -85,B 0,C 180,E1 -19851.408,E2 -19851.408} C_VEL
LIN {X 0,Y 261.725,Z 385.16,A -85,B 0,C 180,E1 -19852.162,E2 -19852.162} C_VEL
LIN {X 0,Y 261.082,Z 389.039,A -85,B 0,C 180,E1 -19853.147,E2 -19853.147} C_VEL
LIN {X 0,Y 259.625,Z 393.478,A -85,B 0,C 180,E1 -19853.998,E2 -19853.998} C_VEL
LIN {X 0,Y 255.944,Z 402.467,A -85,B 0,C 180,E1 -19855.693,E2 -19855.693} C_VEL
LIN {X 0,Y 254.993,Z 405.202,A -85,B 0,C 180,E1 -19856.344,E2 -19856.344} C_VEL
LIN {X 0,Y 252.144,Z 413.386,A -85,B 0,C 180,E1 -19858.492,E2 -19858.492} C_VEL
LIN {X 0,Y 249.317,Z 419.102,A -85,B 0,C 180,E1 -19859.976,E2 -19859.976} C_VEL
LIN {X 0,Y 243.595,Z 427.968,A -85,B 0,C 180,E1 -19862.508,E2 -19862.508} C_VEL
LIN {X 0,Y 239.33,Z 434.172,A -85,B 0,C 180,E1 -19864.799,E2 -19864.799} C_VEL
LIN {X 0,Y 235.542,Z 439.282,A -85,B 0,C 180,E1 -19867.177,E2 -19867.177} C_VEL
LIN {X 0,Y 231.591,Z 444.549,A -85,B 0,C 180,E1 -19870.5,E2 -19870.5} C_VEL
LIN {X 0,Y 228.758,Z 448.282,A -85,B 0,C 180,E1 -19873.948,E2 -19873.948} C_VEL
LIN {X 0,Y 226.908,Z 450.521,A -85,B 0,C 180,E1 -19877.478,E2 -19877.478} C_VEL
LIN {X 0,Y 226.272,Z 451.353,A -85,B 0,C 180,E1 -19881.066,E2 -19881.066} C_VEL
LIN {X 0,Y 226.497,Z 450.701,A -85,B 0,C 180,E1 -19884.659,E2 -19884.659} C_VEL
LIN {X 0,Y 226.822,Z 449.801,A -85,B 0,C 180,E1 -19886.447,E2 -19886.447} C_VEL
LIN {X 0,Y 227.308,Z 448.461,A -85,B 0,C 180,E1 -19888.228,E2 -19888.228} C_VEL
LIN {X 0,Y 227.786,Z 445.524,A -85,B 0,C 180,E1 -19890.884,E2 -19890.884} C_VEL
LIN {X 0,Y 227.886,Z 444.679,A -85,B 0,C 180,E1 -19891.546,E2 -19891.546} C_VEL
LIN {X 0,Y 227.146,Z 447.211,A -85,B 0,C 180,E1 -19893.548,E2 -19893.548} C_VEL
LIN {X 0,Y 226.684,Z 448.755,A -85,B 0,C 180,E1 -19895.337,E2 -19895.337} C_VEL
LIN {X 0,Y 226.465,Z 449.677,A -85,B 0,C 180,E1 -19897.131,E2 -19897.131} C_VEL
LIN {X 0,Y 226.486,Z 450.022,A -85,B 0,C 180,E1 -19898.926,E2 -19898.926} C_VEL
LIN {X 0,Y 226.759,Z 449.803,A -85,B 0,C 180,E1 -19900.717,E2 -19900.717} C_VEL
LIN {X 0,Y 227.374,Z 449.022,A -85,B 0,C 180,E1 -19902.496,E2 -19902.496} C_VEL
LIN {X 0,Y 228.244,Z 447.678,A -85,B 0,C 180,E1 -19904.261,E2 -19904.261} C_VEL
LIN {X 0,Y 230.281,Z 444.534,A -85,B 0,C 180,E1 -19906.854,E2 -19906.854} C_VEL
LIN {X 0,Y 232.915,Z 440.094,A -85,B 0,C 180,E1 -19909.385,E2 -19909.385} C_VEL
LIN {X 0,Y 235.624,Z 435.071,A -85,B 0,C 180,E1 -19911.431,E2 -19911.431} C_VEL
LIN {X 0,Y 238.865,Z 428.829,A -85,B 0,C 180,E1 -19913.404,E2 -19913.404} C_VEL
LIN {X 0,Y 242.471,Z 420.861,A -85,B 0,C 180,E1 -19915.311,E2 -19915.311} C_VEL
LIN {X 0,Y 245.424,Z 413.676,A -85,B 0,C 180,E1 -19916.667,E2 -19916.667} C_VEL
LIN {X 0,Y 247.833,Z 403.564,A -85,B 0,C 180,E1 -19918.464,E2 -19918.464} C_VEL
LIN {X 0,Y 248.542,Z 398.824,A -85,B 0,C 180,E1 -19919.265,E2 -19919.265} C_VEL
LIN {X 0,Y 248.416,Z 388.669,A -85,B 0,C 180,E1 -19921.323,E2 -19921.323} C_VEL
LIN {X 0,Y 247.526,Z 378.349,A -85,B 0,C 180,E1 -19923.606,E2 -19923.606} C_VEL
LIN {X 0,Y 248.559,Z 374.77,A -85,B 0,C 180,E1 -19924.915,E2 -19924.915} C_VEL
LIN {X 0,Y 248.738,Z 372.007,A -85,B 0,C 180,E1 -19926.395,E2 -19926.395} C_VEL
LIN {X 0,Y 248.63,Z 369.092,A -85,B 0,C 180,E1 -19928.453,E2 -19928.453} C_VEL
LIN {X 0,Y 248.172,Z 367.015,A -85,B 0,C 180,E1 -19930.643,E2 -19930.643} C_VEL
LIN {X 0,Y 247.488,Z 365.658,A -85,B 0,C 180,E1 -19932.964,E2 -19932.964} C_VEL
LIN {X 0,Y 246.695,Z 364.993,A -85,B 0,C 180,E1 -19935.416,E2 -19935.416} C_VEL
LIN {X 0,Y 245.698,Z 365.038,A -85,B 0,C 180,E1 -19938.858,E2 -19938.858} C_VEL
LIN {X 0,Y 245.184,Z 365.514,A -85,B 0,C 180,E1 -19940.902,E2 -19940.902} C_VEL
LIN {X 0,Y 244.323,Z 367.191,A -85,B 0,C 180,E1 -19944.599,E2 -19944.599} C_VEL
LIN {X 0,Y 246.134,Z 371.732,A -85,B 0,C 180,E1 -19947.143,E2 -19947.143} C_VEL
LIN {X 0,Y 247.344,Z 376.757,A -85,B 0,C 180,E1 -19949.238,E2 -19949.238} C_VEL
LIN {X 0,Y 248.405,Z 383.066,A -85,B 0,C 180,E1 -19951.666,E2 -19951.666} C_VEL
LIN {X 0,Y 248.986,Z 390.13,A -85,B 0,C 180,E1 -19954.253,E2 -19954.253} C_VEL
LIN {X 0,Y 248.662,Z 396.694,A -85,B 0,C 180,E1 -19956.689,E2 -19956.689} C_VEL
LIN {X 0,Y 248.297,Z 398.877,A -85,B 0,C 180,E1 -19957.533,E2 -19957.533} C_VEL
LIN {X 0,Y 245.629,Z 403.72,A -85,B 0,C 180,E1 -19959.042,E2 -19959.042} C_VEL
LIN {X 0,Y 242.897,Z 407.736,A -85,B 0,C 180,E1 -19960.563,E2 -19960.563} C_VEL
LIN {X 0,Y 240.393,Z 410.845,A -85,B 0,C 180,E1 -19962.121,E2 -19962.121} C_VEL
LIN {X 0,Y 236.993,Z 414.07,A -85,B 0,C 180,E1 -19964.518,E2 -19964.518} C_VEL
LIN {X 0,Y 234.968,Z 415.407,A -85,B 0,C 180,E1 -19966.154,E2 -19966.154} C_VEL
LIN {X 0,Y 233.105,Z 416.097,A -85,B 0,C 180,E1 -19967.814,E2 -19967.814} C_VEL
LIN {X 0,Y 231.324,Z 416.164,A -85,B 0,C 180,E1 -19969.495,E2 -19969.495} C_VEL
LIN {X 0,Y 229.842,Z 415.58,A -85,B 0,C 180,E1 -19971.204,E2 -19971.204} C_VEL
LIN {X 0,Y 228.647,Z 414.348,A -85,B 0,C 180,E1 -19972.935,E2 -19972.935} C_VEL
LIN {X 0,Y 227.291,Z 411.217,A -85,B 0,C 180,E1 -19975.564,E2 -19975.564} C_VEL
LIN {X 0,Y 226.75,Z 408.282,A -85,B 0,C 180,E1 -19977.333,E2 -19977.333} C_VEL
LIN {X 0,Y 226.359,Z 403.577,A -85,B 0,C 180,E1 -19979.553,E2 -19979.553} C_VEL
LIN {X 0,Y 226.329,Z 397.312,A -85,B 0,C 180,E1 -19981.777,E2 -19981.777} C_VEL
LIN {X 0,Y 226.643,Z 389.256,A -85,B 0,C 180,E1 -19983.998,E2 -19983.998} C_VEL
LIN {X 0,Y 227.028,Z 381.047,A -85,B 0,C 180,E1 -19985.772,E2 -19985.772} C_VEL
LIN {X 0,Y 227.265,Z 371.806,A -85,B 0,C 180,E1 -19987.298,E2 -19987.298} C_VEL
LIN {X 0,Y 227.571,Z 361.085,A -85,B 0,C 180,E1 -19988.628,E2 -19988.628} C_VEL
LIN {X 0,Y 227.441,Z 354.578,A -85,B 0,C 180,E1 -19989.238,E2 -19989.238} C_VEL
LIN {X 0,Y 227.159,Z 341.491,A -85,B 0,C 180,E1 -19996.165,E2 -19996.165} C_VEL
LIN {X 0,Y 227.394,Z 332.865,A -85,B 0,C 180,E1 -20000.817,E2 -20000.817} C_VEL
LIN {X 0,Y 227.739,Z 324.07,A -85,B 0,C 180,E1 -20005.594,E2 -20005.594} C_VEL
LIN {X 0,Y 228.136,Z 316.066,A -85,B 0,C 180,E1 -20010.098,E2 -20010.098} C_VEL
LIN {X 0,Y 227.879,Z 316.097,A -85,B 0,C 180,E1 -20015.869,E2 -20015.869} C_VEL
LIN {X 0,Y 227.8,Z 316.107,A -85,B 0,C 180,E1 -20020.379,E2 -20020.379} C_VEL
LIN {X 0,Y 227.818,Z 316.108,A -85,B 0,C 180,E1 -20025.193,E2 -20025.193} C_VEL
LIN {X 0,Y 227.817,Z 316.104,A -85,B 0,C 180,E1 -20029.621,E2 -20029.621} C_VEL
LIN {X 0,Y 227.872,Z 316.098,A -85,B 0,C 180,E1 -20034.126,E2 -20034.126} C_VEL
LIN {X 0,Y 227.862,Z 316.101,A -85,B 0,C 180,E1 -20038.376,E2 -20038.376} C_VEL
LIN {X 0,Y 227.877,Z 316.099,A -85,B 0,C 180,E1 -20042.444,E2 -20042.444} C_VEL
LIN {X 0,Y 227.905,Z 316.097,A -85,B 0,C 180,E1 -20046.366,E2 -20046.366} C_VEL
LIN {X 0,Y 227.933,Z 316.091,A -85,B 0,C 180,E1 -20050.174,E2 -20050.174} C_VEL
LIN {X 0,Y 228.048,Z 316.078,A -85,B 0,C 180,E1 -20053.897,E2 -20053.897} C_VEL
LIN {X 0,Y 228.052,Z 316.073,A -85,B 0,C 180,E1 -20057.542,E2 -20057.542} C_VEL
LIN {X 0,Y 228.246,Z 316.052,A -85,B 0,C 180,E1 -20061.144,E2 -20061.144} C_VEL
LIN {X 0,Y 228.295,Z 316.045,A -85,B 0,C 180,E1 -20062.927,E2 -20062.927} C_VEL
LIN {X 0,Y 228.524,Z 316.02,A -85,B 0,C 180,E1 -20068.238,E2 -20068.238} C_VEL
LIN {X 0,Y 228.524,Z 316.02,A -85,B 0,C 180,E1 -20071.762,E2 -20071.762} C_VEL
LIN {X 0,Y 228.295,Z 316.045,A -85,B 0,C 180,E1 -20077.073,E2 -20077.073} C_VEL
LIN {X 0,Y 228.132,Z 316.065,A -85,B 0,C 180,E1 -20080.652,E2 -20080.652} C_VEL
LIN {X 0,Y 228.047,Z 316.076,A -85,B 0,C 180,E1 -20084.273,E2 -20084.273} C_VEL
LIN {X 0,Y 227.997,Z 316.084,A -85,B 0,C 180,E1 -20087.954,E2 -20087.954} C_VEL
LIN {X 0,Y 227.951,Z 316.087,A -85,B 0,C 180,E1 -20092.349,E2 -20092.349} C_VEL
LIN {X 0,Y 227.934,Z 316.091,A -85,B 0,C 180,E1 -20096.604,E2 -20096.604} C_VEL
LIN {X 0,Y 227.9,Z 316.092,A -85,B 0,C 180,E1 -20100.298,E2 -20100.298} C_VEL
LIN {X 0,Y 227.868,Z 316.1,A -85,B 0,C 180,E1 -20103.722,E2 -20103.722} C_VEL
LIN {X 0,Y 227.836,Z 316.1,A -85,B 0,C 180,E1 -20108.093,E2 -20108.093} C_VEL
LIN {X 0,Y 227.798,Z 316.109,A -85,B 0,C 180,E1 -20112.746,E2 -20112.746} C_VEL
LIN {X 0,Y 227.793,Z 316.108,A -85,B 0,C 180,E1 -20117.257,E2 -20117.257} C_VEL
LIN {X 0,Y 227.84,Z 316.102,A -85,B 0,C 180,E1 -20121.912,E2 -20121.912} C_VEL
LIN {X 0,Y 228.152,Z 316.063,A -85,B 0,C 180,E1 -20127.383,E2 -20127.383} C_VEL
LIN {X 0,Y 228.233,Z 316.189,A -85,B 0,C 180,E1 -20128.178,E2 -20128.178} C_VEL
LIN {X 0,Y 228.13,Z 318.992,A -85,B 0,C 180,E1 -20130.471,E2 -20130.471} C_VEL
LIN {X 0,Y 227.471,Z 325.122,A -85,B 0,C 180,E1 -20135.351,E2 -20135.351} C_VEL
LIN {X 0,Y 226.951,Z 331.201,A -85,B 0,C 180,E1 -20140.087,E2 -20140.087} C_VEL
LIN {X 0,Y 226.55,Z 337.421,A -85,B 0,C 180,E1 -20144.846,E2 -20144.846} C_VEL
LIN {X 0,Y 226.465,Z 340.752,A -85,B 0,C 180,E1 -20147.342,E2 -20147.342} C_VEL
LIN {X 0,Y 227.585,Z 353.506,A -85,B 0,C 180,E1 -20148.649,E2 -20148.649} C_VEL
LIN {X 0,Y 228.058,Z 359.099,A -85,B 0,C 180,E1 -20149.347,E2 -20149.347} C_VEL
LIN {X 0,Y 227.532,Z 370.706,A -85,B 0,C 180,E1 -20151.118,E2 -20151.118} C_VEL
LIN {X 0,Y 227.021,Z 380.986,A -85,B 0,C 180,E1 -20153.113,E2 -20153.113} C_VEL
LIN {X 0,Y 226.716,Z 389.222,A -85,B 0,C 180,E1 -20155.112,E2 -20155.112} C_VEL
LIN {X 0,Y 226.3,Z 397.895,A -85,B 0,C 180,E1 -20157.778,E2 -20157.778} C_VEL
LIN {X 0,Y 226.325,Z 403.653,A -85,B 0,C 180,E1 -20160.002,E2 -20160.002} C_VEL
LIN {X 0,Y 226.765,Z 409.03,A -85,B 0,C 180,E1 -20162.667,E2 -20162.667} C_VEL
LIN {X 0,Y 227.685,Z 412.935,A -85,B 0,C 180,E1 -20165.316,E2 -20165.316} C_VEL
LIN {X 0,Y 228.645,Z 414.827,A -85,B 0,C 180,E1 -20167.065,E2 -20167.065} C_VEL
LIN {X 0,Y 229.779,Z 416.134,A -85,B 0,C 180,E1 -20168.799,E2 -20168.799} C_VEL
LIN {X 0,Y 231.182,Z 416.881,A -85,B 0,C 180,E1 -20170.512,E2 -20170.512} C_VEL
LIN {X 0,Y 232.968,Z 417.089,A -85,B 0,C 180,E1 -20172.193,E2 -20172.193} C_VEL
LIN {X 0,Y 234.848,Z 416.746,A -85,B 0,C 180,E1 -20173.854,E2 -20173.854} C_VEL
LIN {X 0,Y 236.979,Z 415.867,A -85,B 0,C 180,E1 -20175.483,E2 -20175.483} C_VEL
LIN {X 0,Y 239.294,Z 414.507,A -85,B 0,C 180,E1 -20177.082,E2 -20177.082} C_VEL
LIN {X 0,Y 243.14,Z 411.392,A -85,B 0,C 180,E1 -20179.417,E2 -20179.417} C_VEL
LIN {X 0,Y 247.498,Z 406.989,A -85,B 0,C 180,E1 -20181.665,E2 -20181.665} C_VEL
LIN {X 0,Y 250.59,Z 403.327,A -85,B 0,C 180,E1 -20183.121,E2 -20183.121} C_VEL
LIN {X 0,Y 252.038,Z 399.923,A -85,B 0,C 180,E1 -20184.727,E2 -20184.727} C_VEL
LIN {X 0,Y 253.401,Z 394.525,A -85,B 0,C 180,E1 -20187.438,E2 -20187.438} C_VEL
LIN {X 0,Y 254.205,Z 388.864,A -85,B 0,C 180,E1 -20190.441,E2 -20190.441} C_VEL
LIN {X 0,Y 254.513,Z 385.282,A -85,B 0,C 180,E1 -20192.636,E2 -20192.636} C_VEL
LIN {X 0,Y 254.332,Z 381.995,A -85,B 0,C 180,E1 -20195.473,E2 -20195.473} C_VEL
LIN {X 0,Y 254.09,Z 380.686,A -85,B 0,C 180,E1 -20197.484,E2 -20197.484} C_VEL
LIN {X 0,Y 253.878,Z 380.07,A -85,B 0,C 180,E1 -20199.548,E2 -20199.548} C_VEL
LIN {X 0,Y 253.929,Z 380.049,A -85,B 0,C 180,E1 -20201.644,E2 -20201.644} C_VEL
LIN {X 0,Y 254.276,Z 380.915,A -85,B 0,C 180,E1 -20204.059,E2 -20204.059} C_VEL
LIN {X 0,Y 254.941,Z 382.629,A -85,B 0,C 180,E1 -20206.435,E2 -20206.435} C_VEL
LIN {X 0,Y 256.118,Z 385.006,A -85,B 0,C 180,E1 -20208.809,E2 -20208.809} C_VEL
LIN {X 0,Y 257.818,Z 390.76,A -85,B 0,C 180,E1 -20212.237,E2 -20212.237} C_VEL
LIN {X 0,Y 257.792,Z 393.29,A -85,B 0,C 180,E1 -20213.146,E2 -20213.146} C_VEL
LIN {X 0,Y 255.522,Z 403.336,A -85,B 0,C 180,E1 -20215.858,E2 -20215.858} C_VEL
LIN {X 0,Y 254.993,Z 405.202,A -85,B 0,C 180,E1 -20216.344,E2 -20216.344} C_VEL
LIN {X 0,Y 253.928,Z 407.855,A -85,B 0,C 180,E1 -20216.965,E2 -20216.965} C_VEL
LIN {X 0,Y 252.366,Z 410.626,A -85,B 0,C 180,E1 -20217.508,E2 -20217.508} C_VEL
LIN {X 0,Y 248.298,Z 416.135,A -85,B 0,C 180,E1 -20218.463,E2 -20218.463} C_VEL
LIN {X 0,Y 243.758,Z 421.319,A -85,B 0,C 180,E1 -20219.435,E2 -20219.435} C_VEL
LIN {X 0,Y 240.669,Z 424.887,A -85,B 0,C 180,E1 -20220.314,E2 -20220.314} C_VEL
LIN {X 0,Y 239.799,Z 425.998,A -85,B 0,C 180,E1 -20220.653,E2 -20220.653} C_VEL
LIN {X 0,Y 235.818,Z 431.262,A -85,B 0,C 180,E1 -20222.487,E2 -20222.487} C_VEL
LIN {X 0,Y 230.284,Z 438.236,A -85,B 0,C 180,E1 -20225.669,E2 -20225.669} C_VEL
LIN {X 0,Y 225.89,Z 443.407,A -85,B 0,C 180,E1 -20228.972,E2 -20228.972} C_VEL
LIN {X 0,Y 223.276,Z 446.411,A -85,B 0,C 180,E1 -20231.653,E2 -20231.653} C_VEL
LIN {X 0,Y 220.803,Z 449.062,A -85,B 0,C 180,E1 -20235.248,E2 -20235.248} C_VEL
LIN {X 0,Y 219.516,Z 450.265,A -85,B 0,C 180,E1 -20238.925,E2 -20238.925} C_VEL
LIN {X 0,Y 219.247,Z 450.082,A -85,B 0,C 180,E1 -20242.633,E2 -20242.633} C_VEL
LIN {X 0,Y 219.512,Z 449.427,A -85,B 0,C 180,E1 -20244.488,E2 -20244.488} C_VEL
LIN {X 0,Y 220.361,Z 446.935,A -85,B 0,C 180,E1 -20248.172,E2 -20248.172} C_VEL
LIN {X 0,Y 220.883,Z 443.774,A -85,B 0,C 180,E1 -20250.912,E2 -20250.912} C_VEL
LIN {X 0,Y 221.033,Z 442.803,A -85,B 0,C 180,E1 -20251.651,E2 -20251.651} C_VEL
LIN {X 0,Y 220.264,Z 445.516,A -85,B 0,C 180,E1 -20253.659,E2 -20253.659} C_VEL
LIN {X 0,Y 219.738,Z 447.249,A -85,B 0,C 180,E1 -20255.506,E2 -20255.506} C_VEL
LIN {X 0,Y 219.505,Z 448.391,A -85,B 0,C 180,E1 -20257.358,E2 -20257.358} C_VEL
LIN {X 0,Y 219.497,Z 448.953,A -85,B 0,C 180,E1 -20259.212,E2 -20259.212} C_VEL
LIN {X 0,Y 219.78,Z 448.956,A -85,B 0,C 180,E1 -20261.062,E2 -20261.062} C_VEL
LIN {X 0,Y 220.442,Z 448.425,A -85,B 0,C 180,E1 -20262.895,E2 -20262.895} C_VEL
LIN {X 0,Y 221.35,Z 447.336,A -85,B 0,C 180,E1 -20264.715,E2 -20264.715} C_VEL
LIN {X 0,Y 223.513,Z 444.716,A -85,B 0,C 180,E1 -20267.38,E2 -20267.38} C_VEL
LIN {X 0,Y 226.271,Z 440.654,A -85,B 0,C 180,E1 -20269.978,E2 -20269.978} C_VEL
LIN {X 0,Y 229.761,Z 435.204,A -85,B 0,C 180,E1 -20272.48,E2 -20272.48} C_VEL
LIN {X 0,Y 233.928,Z 427.856,A -85,B 0,C 180,E1 -20274.873,E2 -20274.873} C_VEL
LIN {X 0,Y 237.929,Z 420.063,A -85,B 0,C 180,E1 -20276.747,E2 -20276.747} C_VEL
LIN {X 0,Y 240.391,Z 414.31,A -85,B 0,C 180,E1 -20277.89,E2 -20277.89} C_VEL
LIN {X 0,Y 243.273,Z 404.415,A -85,B 0,C 180,E1 -20279.761,E2 -20279.761} C_VEL
LIN {X 0,Y 243.899,Z 399.545,A -85,B 0,C 180,E1 -20280.761,E2 -20280.761} C_VEL
LIN {X 0,Y 244.186,Z 390.401,A -85,B 0,C 180,E1 -20282.776,E2 -20282.776} C_VEL
LIN {X 0,Y 243.747,Z 380.322,A -85,B 0,C 180,E1 -20285.216,E2 -20285.216} C_VEL
LIN {X 0,Y 243.278,Z 377.232,A -85,B 0,C 180,E1 -20286.2,E2 -20286.2} C_VEL
LIN {X 0,Y 243.142,Z 373.487,A -85,B 0,C 180,E1 -20288.697,E2 -20288.697} C_VEL
LIN {X 0,Y 242.314,Z 370.778,A -85,B 0,C 180,E1 -20291.843,E2 -20291.843} C_VEL
LIN {X 0,Y 241.529,Z 369.684,A -85,B 0,C 180,E1 -20294.295,E2 -20294.295} C_VEL
LIN {X 0,Y 240.368,Z 369.263,A -85,B 0,C 180,E1 -20297.739,E2 -20297.739} C_VEL
LIN {X 0,Y 239.65,Z 369.79,A -85,B 0,C 180,E1 -20300.483,E2 -20300.483} C_VEL
LIN {X 0,Y 241.582,Z 374.008,A -85,B 0,C 180,E1 -20304.545,E2 -20304.545} C_VEL
LIN {X 0,Y 242.6,Z 377.433,A -85,B 0,C 180,E1 -20306.602,E2 -20306.602} C_VEL
LIN {X 0,Y 243.262,Z 382,A -85,B 0,C 180,E1 -20308.663,E2 -20308.663} C_VEL
LIN {X 0,Y 243.731,Z 387.743,A -85,B 0,C 180,E1 -20311.072,E2 -20311.072} C_VEL
LIN {X 0,Y 243.702,Z 394.949,A -85,B 0,C 180,E1 -20313.997,E2 -20313.997} C_VEL
LIN {X 0,Y 242.716,Z 401.051,A -85,B 0,C 180,E1 -20316.536,E2 -20316.536} C_VEL
LIN {X 0,Y 242.376,Z 402.136,A -85,B 0,C 180,E1 -20316.953,E2 -20316.953} C_VEL
LIN {X 0,Y 239.367,Z 406.573,A -85,B 0,C 180,E1 -20318.467,E2 -20318.467} C_VEL
LIN {X 0,Y 235.185,Z 411.605,A -85,B 0,C 180,E1 -20320.807,E2 -20320.807} C_VEL
LIN {X 0,Y 232.656,Z 413.999,A -85,B 0,C 180,E1 -20322.415,E2 -20322.415} C_VEL
LIN {X 0,Y 230.34,Z 415.676,A -85,B 0,C 180,E1 -20324.059,E2 -20324.059} C_VEL
LIN {X 0,Y 228.186,Z 416.706,A -85,B 0,C 180,E1 -20325.733,E2 -20325.733} C_VEL
LIN {X 0,Y 226.231,Z 417.117,A -85,B 0,C 180,E1 -20327.438,E2 -20327.438} C_VEL
LIN {X 0,Y 224.382,Z 416.903,A -85,B 0,C 180,E1 -20329.166,E2 -20329.166} C_VEL
LIN {X 0,Y 222.852,Z 416.036,A -85,B 0,C 180,E1 -20330.925,E2 -20330.925} C_VEL
LIN {X 0,Y 221.088,Z 413.556,A -85,B 0,C 180,E1 -20333.61,E2 -20333.61} C_VEL
LIN {X 0,Y 220.214,Z 411.071,A -85,B 0,C 180,E1 -20335.421,E2 -20335.421} C_VEL
LIN {X 0,Y 219.665,Z 407.844,A -85,B 0,C 180,E1 -20337.247,E2 -20337.247} C_VEL
LIN {X 0,Y 219.316,Z 402.63,A -85,B 0,C 180,E1 -20339.539,E2 -20339.539} C_VEL
LIN {X 0,Y 219.306,Z 396.023,A -85,B 0,C 180,E1 -20341.834,E2 -20341.834} C_VEL
LIN {X 0,Y 219.669,Z 387.448,A -85,B 0,C 180,E1 -20344.126,E2 -20344.126} C_VEL
LIN {X 0,Y 220.006,Z 379.633,A -85,B 0,C 180,E1 -20345.727,E2 -20345.727} C_VEL
LIN {X 0,Y 220.291,Z 369.633,A -85,B 0,C 180,E1 -20347.329,E2 -20347.329} C_VEL
LIN {X 0,Y 220.562,Z 359.72,A -85,B 0,C 180,E1 -20348.513,E2 -20348.513} C_VEL
LIN {X 0,Y 220.468,Z 355.191,A -85,B 0,C 180,E1 -20348.968,E2 -20348.968} C_VEL
LIN {X 0,Y 220.051,Z 342.647,A -85,B 0,C 180,E1 -20355.718,E2 -20355.718} C_VEL
LIN {X 0,Y 220.292,Z 333.85,A -85,B 0,C 180,E1 -20360.542,E2 -20360.542} C_VEL
LIN {X 0,Y 220.637,Z 324.93,A -85,B 0,C 180,E1 -20365.466,E2 -20365.466} C_VEL
LIN {X 0,Y 221.041,Z 316.95,A -85,B 0,C 180,E1 -20369.916,E2 -20369.916} C_VEL
LIN {X 0,Y 220.804,Z 316.977,A -85,B 0,C 180,E1 -20374.951,E2 -20374.951} C_VEL
LIN {X 0,Y 220.805,Z 316.982,A -85,B 0,C 180,E1 -20377.276,E2 -20377.276} C_VEL
LIN {X 0,Y 220.752,Z 316.983,A -85,B 0,C 180,E1 -20381.953,E2 -20381.953} C_VEL
LIN {X 0,Y 220.76,Z 316.985,A -85,B 0,C 180,E1 -20385.542,E2 -20385.542} C_VEL
LIN {X 0,Y 220.799,Z 316.979,A -85,B 0,C 180,E1 -20390.461,E2 -20390.461} C_VEL
LIN {X 0,Y 220.792,Z 316.982,A -85,B 0,C 180,E1 -20395.043,E2 -20395.043} C_VEL
LIN {X 0,Y 220.86,Z 316.969,A -85,B 0,C 180,E1 -20399.393,E2 -20399.393} C_VEL
LIN {X 0,Y 220.886,Z 316.969,A -85,B 0,C 180,E1 -20403.548,E2 -20403.548} C_VEL
LIN {X 0,Y 220.869,Z 316.969,A -85,B 0,C 180,E1 -20407.552,E2 -20407.552} C_VEL
LIN {X 0,Y 220.975,Z 316.96,A -85,B 0,C 180,E1 -20412.57,E2 -20412.57} C_VEL
LIN {X 0,Y 220.993,Z 316.952,A -85,B 0,C 180,E1 -20417.137,E2 -20417.137} C_VEL
LIN {X 0,Y 221.186,Z 316.932,A -85,B 0,C 180,E1 -20420.859,E2 -20420.859} C_VEL
LIN {X 0,Y 221.232,Z 316.926,A -85,B 0,C 180,E1 -20422.7,E2 -20422.7} C_VEL
LIN {X 0,Y 221.457,Z 316.9,A -85,B 0,C 180,E1 -20428.181,E2 -20428.181} C_VEL
LIN {X 0,Y 221.457,Z 316.9,A -85,B 0,C 180,E1 -20431.819,E2 -20431.819} C_VEL
LIN {X 0,Y 221.232,Z 316.926,A -85,B 0,C 180,E1 -20437.3,E2 -20437.3} C_VEL
LIN {X 0,Y 221.054,Z 316.947,A -85,B 0,C 180,E1 -20440.997,E2 -20440.997} C_VEL
LIN {X 0,Y 221.007,Z 316.954,A -85,B 0,C 180,E1 -20446.631,E2 -20446.631} C_VEL
LIN {X 0,Y 220.9,Z 316.965,A -85,B 0,C 180,E1 -20450.486,E2 -20450.486} C_VEL
LIN {X 0,Y 220.864,Z 316.971,A -85,B 0,C 180,E1 -20454.436,E2 -20454.436} C_VEL
LIN {X 0,Y 220.828,Z 316.974,A -85,B 0,C 180,E1 -20458.515,E2 -20458.515} C_VEL
LIN {X 0,Y 220.809,Z 316.978,A -85,B 0,C 180,E1 -20462.758,E2 -20462.758} C_VEL
LIN {X 0,Y 220.802,Z 316.979,A -85,B 0,C 180,E1 -20467.28,E2 -20467.28} C_VEL
LIN {X 0,Y 220.787,Z 316.979,A -85,B 0,C 180,E1 -20470.19,E2 -20470.19} C_VEL
LIN {X 0,Y 220.76,Z 316.985,A -85,B 0,C 180,E1 -20474.458,E2 -20474.458} C_VEL
LIN {X 0,Y 220.752,Z 316.983,A -85,B 0,C 180,E1 -20478.047,E2 -20478.047} C_VEL
LIN {X 0,Y 220.819,Z 316.98,A -85,B 0,C 180,E1 -20482.795,E2 -20482.795} C_VEL
LIN {X 0,Y 221.177,Z 316.989,A -85,B 0,C 180,E1 -20488.153,E2 -20488.153} C_VEL
LIN {X 0,Y 221.059,Z 319.767,A -85,B 0,C 180,E1 -20490.479,E2 -20490.479} C_VEL
LIN {X 0,Y 220.385,Z 325.931,A -85,B 0,C 180,E1 -20495.511,E2 -20495.511} C_VEL
LIN {X 0,Y 219.946,Z 330.826,A -85,B 0,C 180,E1 -20499.424,E2 -20499.424} C_VEL
LIN {X 0,Y 219.534,Z 336.43,A -85,B 0,C 180,E1 -20503.822,E2 -20503.822} C_VEL
LIN {X 0,Y 219.402,Z 341.312,A -85,B 0,C 180,E1 -20507.457,E2 -20507.457} C_VEL
LIN {X 0,Y 220.501,Z 353.682,A -85,B 0,C 180,E1 -20508.745,E2 -20508.745} C_VEL
LIN {X 0,Y 220.942,Z 359.305,A -85,B 0,C 180,E1 -20509.464,E2 -20509.464} C_VEL
LIN {X 0,Y 220.474,Z 370.302,A -85,B 0,C 180,E1 -20511.183,E2 -20511.183} C_VEL
LIN {X 0,Y 219.961,Z 381.156,A -85,B 0,C 180,E1 -20513.351,E2 -20513.351} C_VEL
LIN {X 0,Y 219.611,Z 389.423,A -85,B 0,C 180,E1 -20515.414,E2 -20515.414} C_VEL
LIN {X 0,Y 219.211,Z 398.25,A -85,B 0,C 180,E1 -20518.165,E2 -20518.165} C_VEL
LIN {X 0,Y 219.36,Z 405.07,A -85,B 0,C 180,E1 -20520.92,E2 -20520.92} C_VEL
LIN {X 0,Y 219.938,Z 410.272,A -85,B 0,C 180,E1 -20523.667,E2 -20523.667} C_VEL
LIN {X 0,Y 221.097,Z 414.075,A -85,B 0,C 180,E1 -20526.39,E2 -20526.39} C_VEL
LIN {X 0,Y 222.794,Z 416.59,A -85,B 0,C 180,E1 -20529.077,E2 -20529.077} C_VEL
LIN {X 0,Y 224.251,Z 417.568,A -85,B 0,C 180,E1 -20530.841,E2 -20530.841} C_VEL
LIN {X 0,Y 226.079,Z 417.991,A -85,B 0,C 180,E1 -20532.571,E2 -20532.571} C_VEL
LIN {X 0,Y 228.067,Z 417.912,A -85,B 0,C 180,E1 -20534.274,E2 -20534.274} C_VEL
LIN {X 0,Y 230.276,Z 417.287,A -85,B 0,C 180,E1 -20535.945,E2 -20535.945} C_VEL
LIN {X 0,Y 232.687,Z 416.152,A -85,B 0,C 180,E1 -20537.582,E2 -20537.582} C_VEL
LIN {X 0,Y 236.688,Z 413.476,A -85,B 0,C 180,E1 -20539.969,E2 -20539.969} C_VEL
LIN {X 0,Y 241.231,Z 409.535,A -85,B 0,C 180,E1 -20542.258,E2 -20542.258} C_VEL
LIN {X 0,Y 244.419,Z 406.186,A -85,B 0,C 180,E1 -20543.74,E2 -20543.74} C_VEL
LIN {X 0,Y 245.579,Z 404.565,A -85,B 0,C 180,E1 -20544.519,E2 -20544.519} C_VEL
LIN {X 0,Y 247.406,Z 400.01,A -85,B 0,C 180,E1 -20547.035,E2 -20547.035} C_VEL
LIN {X 0,Y 248.684,Z 395.51,A -85,B 0,C 180,E1 -20549.614,E2 -20549.614} C_VEL
LIN {X 0,Y 249.573,Z 391.198,A -85,B 0,C 180,E1 -20552.349,E2 -20552.349} C_VEL
LIN {X 0,Y 249.843,Z 388.853,A -85,B 0,C 180,E1 -20554.238,E2 -20554.238} C_VEL
LIN {X 0,Y 249.868,Z 387.116,A -85,B 0,C 180,E1 -20556.206,E2 -20556.206} C_VEL
LIN {X 0,Y 249.757,Z 386.14,A -85,B 0,C 180,E1 -20558.25,E2 -20558.25} C_VEL
LIN {X 0,Y 249.767,Z 385.853,A -85,B 0,C 180,E1 -20560.559,E2 -20560.559} C_VEL
LIN {X 0,Y 250.044,Z 386.335,A -85,B 0,C 180,E1 -20563.048,E2 -20563.048} C_VEL
LIN {X 0,Y 250.58,Z 387.735,A -85,B 0,C 180,E1 -20565.478,E2 -20565.478} C_VEL
LIN {X 0,Y 251.468,Z 389.815,A -85,B 0,C 180,E1 -20567.875,E2 -20567.875} C_VEL
LIN {X 0,Y 251.885,Z 390.989,A -85,B 0,C 180,E1 -20568.883,E2 -20568.883} C_VEL
LIN {X 0,Y 252.895,Z 395.119,A -85,B 0,C 180,E1 -20571.505,E2 -20571.505} C_VEL
LIN {X 0,Y 252.927,Z 396.949,A -85,B 0,C 180,E1 -20572.316,E2 -20572.316} C_VEL
LIN {X 0,Y 250.619,Z 404.972,A -85,B 0,C 180,E1 -20574.657,E2 -20574.657} C_VEL
LIN {X 0,Y 247.671,Z 412.842,A -85,B 0,C 180,E1 -20576.89,E2 -20576.89} C_VEL
LIN {X 0,Y 244.215,Z 419.623,A -85,B 0,C 180,E1 -20578.801,E2 -20578.801} C_VEL
LIN {X 0,Y 239.799,Z 425.998,A -85,B 0,C 180,E1 -20580.653,E2 -20580.653} C_VEL
LIN {X 0,Y 236.866,Z 429.262,A -85,B 0,C 180,E1 -20581.63,E2 -20581.63} C_VEL
LIN {X 0,Y 230.67,Z 434.178,A -85,B 0,C 180,E1 -20583.117,E2 -20583.117} C_VEL
LIN {X 0,Y 224.718,Z 438.333,A -85,B 0,C 180,E1 -20584.782,E2 -20584.782} C_VEL
LIN {X 0,Y 222.213,Z 440.446,A -85,B 0,C 180,E1 -20586.02,E2 -20586.02} C_VEL
LIN {X 0,Y 218.225,Z 444.51,A -85,B 0,C 180,E1 -20589.252,E2 -20589.252} C_VEL
LIN {X 0,Y 215.071,Z 447.474,A -85,B 0,C 180,E1 -20592.896,E2 -20592.896} C_VEL
LIN {X 0,Y 213.019,Z 449.068,A -85,B 0,C 180,E1 -20596.647,E2 -20596.647} C_VEL
LIN {X 0,Y 212.297,Z 449.268,A -85,B 0,C 180,E1 -20600.472,E2 -20600.472} C_VEL
LIN {X 0,Y 212.519,Z 448.069,A -85,B 0,C 180,E1 -20604.306,E2 -20604.306} C_VEL
LIN {X 0,Y 212.918,Z 446.887,A -85,B 0,C 180,E1 -20606.215,E2 -20606.215} C_VEL
LIN {X 0,Y 213.624,Z 444.28,A -85,B 0,C 180,E1 -20609.057,E2 -20609.057} C_VEL
LIN {X 0,Y 214.22,Z 440.878,A -85,B 0,C 180,E1 -20611.763,E2 -20611.763} C_VEL
LIN {X 0,Y 213.394,Z 443.697,A -85,B 0,C 180,E1 -20613.777,E2 -20613.777} C_VEL
LIN {X 0,Y 212.81,Z 445.671,A -85,B 0,C 180,E1 -20615.686,E2 -20615.686} C_VEL
LIN {X 0,Y 212.538,Z 447.03,A -85,B 0,C 180,E1 -20617.601,E2 -20617.601} C_VEL
LIN {X 0,Y 212.522,Z 447.82,A -85,B 0,C 180,E1 -20619.517,E2 -20619.517} C_VEL
LIN {X 0,Y 212.818,Z 448.078,A -85,B 0,C 180,E1 -20621.428,E2 -20621.428} C_VEL
LIN {X 0,Y 213.526,Z 447.804,A -85,B 0,C 180,E1 -20623.321,E2 -20623.321} C_VEL
LIN {X 0,Y 214.472,Z 446.98,A -85,B 0,C 180,E1 -20625.198,E2 -20625.198} C_VEL
LIN {X 0,Y 215.886,Z 445.62,A -85,B 0,C 180,E1 -20627.037,E2 -20627.037} C_VEL
LIN {X 0,Y 218.606,Z 442.501,A -85,B 0,C 180,E1 -20629.729,E2 -20629.729} C_VEL
LIN {X 0,Y 221.969,Z 438.085,A -85,B 0,C 180,E1 -20632.33,E2 -20632.33} C_VEL
LIN {X 0,Y 225.401,Z 433.177,A -85,B 0,C 180,E1 -20634.402,E2 -20634.402} C_VEL
LIN {X 0,Y 229.258,Z 427.016,A -85,B 0,C 180,E1 -20636.392,E2 -20636.392} C_VEL
LIN {X 0,Y 233.675,Z 419.222,A -85,B 0,C 180,E1 -20638.275,E2 -20638.275} C_VEL
LIN {X 0,Y 236.307,Z 412.839,A -85,B 0,C 180,E1 -20639.67,E2 -20639.67} C_VEL
LIN {X 0,Y 238.71,Z 405.746,A -85,B 0,C 180,E1 -20641.064,E2 -20641.064} C_VEL
LIN {X 0,Y 239.863,Z 396.417,A -85,B 0,C 180,E1 -20643.26,E2 -20643.26} C_VEL
LIN {X 0,Y 240.239,Z 388.423,A -85,B 0,C 180,E1 -20645.279,E2 -20645.279} C_VEL
LIN {X 0,Y 240.298,Z 383.69,A -85,B 0,C 180,E1 -20646.58,E2 -20646.58} C_VEL
LIN {X 0,Y 239.179,Z 379.732,A -85,B 0,C 180,E1 -20648.638,E2 -20648.638} C_VEL
LIN {X 0,Y 238.238,Z 377.421,A -85,B 0,C 180,E1 -20650.466,E2 -20650.466} C_VEL
LIN {X 0,Y 237.266,Z 375.555,A -85,B 0,C 180,E1 -20652.944,E2 -20652.944} C_VEL
LIN {X 0,Y 236.696,Z 374.963,A -85,B 0,C 180,E1 -20655.448,E2 -20655.448} C_VEL
LIN {X 0,Y 236.605,Z 375.348,A -85,B 0,C 180,E1 -20657.953,E2 -20657.953} C_VEL
LIN {X 0,Y 237.073,Z 376.483,A -85,B 0,C 180,E1 -20660.423,E2 -20660.423} C_VEL
LIN {X 0,Y 238.117,Z 379.677,A -85,B 0,C 180,E1 -20663.82,E2 -20663.82} C_VEL
LIN {X 0,Y 238.751,Z 382.875,A -85,B 0,C 180,E1 -20665.991,E2 -20665.991} C_VEL
LIN {X 0,Y 238.955,Z 386.942,A -85,B 0,C 180,E1 -20668.033,E2 -20668.033} C_VEL
LIN {X 0,Y 238.847,Z 393.043,A -85,B 0,C 180,E1 -20670.815,E2 -20670.815} C_VEL
LIN {X 0,Y 238.28,Z 398.589,A -85,B 0,C 180,E1 -20673.335,E2 -20673.335} C_VEL
LIN {X 0,Y 237.216,Z 403.333,A -85,B 0,C 180,E1 -20675.493,E2 -20675.493} C_VEL
LIN {X 0,Y 236.291,Z 405.227,A -85,B 0,C 180,E1 -20676.324,E2 -20676.324} C_VEL
LIN {X 0,Y 233.093,Z 409.261,A -85,B 0,C 180,E1 -20677.857,E2 -20677.857} C_VEL
LIN {X 0,Y 230.149,Z 412.449,A -85,B 0,C 180,E1 -20679.439,E2 -20679.439} C_VEL
LIN {X 0,Y 227.384,Z 414.854,A -85,B 0,C 180,E1 -20681.06,E2 -20681.06} C_VEL
LIN {X 0,Y 223.665,Z 417.113,A -85,B 0,C 180,E1 -20683.57,E2 -20683.57} C_VEL
LIN {X 0,Y 221.404,Z 417.871,A -85,B 0,C 180,E1 -20685.287,E2 -20685.287} C_VEL
LIN {X 0,Y 219.349,Z 417.999,A -85,B 0,C 180,E1 -20687.037,E2 -20687.037} C_VEL
LIN {X 0,Y 217.45,Z 417.505,A -85,B 0,C 180,E1 -20688.816,E2 -20688.816} C_VEL
LIN {X 0,Y 215.87,Z 416.373,A -85,B 0,C 180,E1 -20690.629,E2 -20690.629} C_VEL
LIN {X 0,Y 214.029,Z 413.464,A -85,B 0,C 180,E1 -20693.398,E2 -20693.398} C_VEL
LIN {X 0,Y 212.815,Z 409.047,A -85,B 0,C 180,E1 -20696.211,E2 -20696.211} C_VEL
LIN {X 0,Y 212.373,Z 403.995,A -85,B 0,C 180,E1 -20698.575,E2 -20698.575} C_VEL
LIN {X 0,Y 212.253,Z 397.531,A -85,B 0,C 180,E1 -20700.946,E2 -20700.946} C_VEL
LIN {X 0,Y 212.466,Z 390.981,A -85,B 0,C 180,E1 -20702.842,E2 -20702.842} C_VEL
LIN {X 0,Y 212.9,Z 382.998,A -85,B 0,C 180,E1 -20704.731,E2 -20704.731} C_VEL
LIN {X 0,Y 213.086,Z 373.855,A -85,B 0,C 180,E1 -20706.389,E2 -20706.389} C_VEL
LIN {X 0,Y 213.407,Z 363.809,A -85,B 0,C 180,E1 -20707.773,E2 -20707.773} C_VEL
LIN {X 0,Y 213.528,Z 355.903,A -85,B 0,C 180,E1 -20708.603,E2 -20708.603} C_VEL
LIN {X 0,Y 212.972,Z 342.253,A -85,B 0,C 180,E1 -20716.09,E2 -20716.09} C_VEL
LIN {X 0,Y 213.249,Z 333.014,A -85,B 0,C 180,E1 -20721.252,E2 -20721.252} C_VEL
LIN {X 0,Y 213.634,Z 323.967,A -85,B 0,C 180,E1 -20726.352,E2 -20726.352} C_VEL
LIN {X 0,Y 213.97,Z 317.831,A -85,B 0,C 180,E1 -20729.92,E2 -20729.92} C_VEL
LIN {X 0,Y 213.777,Z 317.851,A -85,B 0,C 180,E1 -20734.726,E2 -20734.726} C_VEL
LIN {X 0,Y 213.703,Z 317.865,A -85,B 0,C 180,E1 -20738.667,E2 -20738.667} C_VEL
LIN {X 0,Y 213.696,Z 317.863,A -85,B 0,C 180,E1 -20743.653,E2 -20743.653} C_VEL
LIN {X 0,Y 213.696,Z 317.865,A -85,B 0,C 180,E1 -20746.343,E2 -20746.343} C_VEL
LIN {X 0,Y 213.709,Z 317.863,A -85,B 0,C 180,E1 -20749.141,E2 -20749.141} C_VEL
LIN {X 0,Y 213.735,Z 317.859,A -85,B 0,C 180,E1 -20753.71,E2 -20753.71} C_VEL
LIN {X 0,Y 213.787,Z 317.853,A -85,B 0,C 180,E1 -20758.723,E2 -20758.723} C_VEL
LIN {X 0,Y 213.817,Z 317.852,A -85,B 0,C 180,E1 -20762.602,E2 -20762.602} C_VEL
LIN {X 0,Y 213.843,Z 317.845,A -85,B 0,C 180,E1 -20766.951,E2 -20766.951} C_VEL
LIN {X 0,Y 213.923,Z 317.839,A -85,B 0,C 180,E1 -20772.304,E2 -20772.304} C_VEL
LIN {X 0,Y 213.936,Z 317.832,A -85,B 0,C 180,E1 -20776.705,E2 -20776.705} C_VEL
LIN {X 0,Y 214.125,Z 317.813,A -85,B 0,C 180,E1 -20780.554,E2 -20780.554} C_VEL
LIN {X 0,Y 214.066,Z 317.818,A -85,B 0,C 180,E1 -20784.348,E2 -20784.348} C_VEL
LIN {X 0,Y 214.394,Z 317.78,A -85,B 0,C 180,E1 -20788.121,E2 -20788.121} C_VEL
LIN {X 0,Y 214.501,Z 317.768,A -85,B 0,C 180,E1 -20790,E2 -20790} C_VEL
LIN {X 0,Y 214.394,Z 317.78,A -85,B 0,C 180,E1 -20791.879,E2 -20791.879} C_VEL
LIN {X 0,Y 214.174,Z 317.806,A -85,B 0,C 180,E1 -20797.542,E2 -20797.542} C_VEL
LIN {X 0,Y 213.985,Z 317.829,A -85,B 0,C 180,E1 -20801.365,E2 -20801.365} C_VEL
LIN {X 0,Y 213.92,Z 317.836,A -85,B 0,C 180,E1 -20805.238,E2 -20805.238} C_VEL
LIN {X 0,Y 213.866,Z 317.844,A -85,B 0,C 180,E1 -20809.185,E2 -20809.185} C_VEL
LIN {X 0,Y 213.846,Z 317.845,A -85,B 0,C 180,E1 -20813.227,E2 -20813.227} C_VEL
LIN {X 0,Y 213.82,Z 317.851,A -85,B 0,C 180,E1 -20817.451,E2 -20817.451} C_VEL
LIN {X 0,Y 213.768,Z 317.856,A -85,B 0,C 180,E1 -20821.738,E2 -20821.738} C_VEL
LIN {X 0,Y 213.735,Z 317.859,A -85,B 0,C 180,E1 -20826.29,E2 -20826.29} C_VEL
LIN {X 0,Y 213.703,Z 317.866,A -85,B 0,C 180,E1 -20831.128,E2 -20831.128} C_VEL
LIN {X 0,Y 213.696,Z 317.865,A -85,B 0,C 180,E1 -20833.681,E2 -20833.681} C_VEL
LIN {X 0,Y 213.696,Z 317.863,A -85,B 0,C 180,E1 -20836.347,E2 -20836.347} C_VEL
LIN {X 0,Y 213.714,Z 317.863,A -85,B 0,C 180,E1 -20841.335,E2 -20841.335} C_VEL
LIN {X 0,Y 214.042,Z 317.821,A -85,B 0,C 180,E1 -20847.199,E2 -20847.199} C_VEL
LIN {X 0,Y 214.171,Z 318.005,A -85,B 0,C 180,E1 -20848.332,E2 -20848.332} C_VEL
LIN {X 0,Y 213.832,Z 321.769,A -85,B 0,C 180,E1 -20851.542,E2 -20851.542} C_VEL
LIN {X 0,Y 213.168,Z 327.958,A -85,B 0,C 180,E1 -20856.698,E2 -20856.698} C_VEL
LIN {X 0,Y 212.616,Z 334.104,A -85,B 0,C 180,E1 -20861.701,E2 -20861.701} C_VEL
LIN {X 0,Y 212.293,Z 340.858,A -85,B 0,C 180,E1 -20867.09,E2 -20867.09} C_VEL
LIN {X 0,Y 212.303,Z 341.397,A -85,B 0,C 180,E1 -20867.516,E2 -20867.516} C_VEL
LIN {X 0,Y 213.585,Z 355.552,A -85,B 0,C 180,E1 -20869.096,E2 -20869.096} C_VEL
LIN {X 0,Y 213.801,Z 360.836,A -85,B 0,C 180,E1 -20869.826,E2 -20869.826} C_VEL
LIN {X 0,Y 213.28,Z 372.019,A -85,B 0,C 180,E1 -20871.689,E2 -20871.689} C_VEL
LIN {X 0,Y 212.865,Z 382.279,A -85,B 0,C 180,E1 -20873.843,E2 -20873.843} C_VEL
LIN {X 0,Y 212.41,Z 391.281,A -85,B 0,C 180,E1 -20876.208,E2 -20876.208} C_VEL
LIN {X 0,Y 212.175,Z 399.734,A -85,B 0,C 180,E1 -20879.054,E2 -20879.054} C_VEL
LIN {X 0,Y 212.391,Z 406.372,A -85,B 0,C 180,E1 -20881.899,E2 -20881.899} C_VEL
LIN {X 0,Y 213.204,Z 411.481,A -85,B 0,C 180,E1 -20884.729,E2 -20884.729} C_VEL
LIN {X 0,Y 214.563,Z 415.154,A -85,B 0,C 180,E1 -20887.531,E2 -20887.531} C_VEL
LIN {X 0,Y 215.816,Z 416.916,A -85,B 0,C 180,E1 -20889.373,E2 -20889.373} C_VEL
LIN {X 0,Y 217.329,Z 418.157,A -85,B 0,C 180,E1 -20891.19,E2 -20891.19} C_VEL
LIN {X 0,Y 219.194,Z 418.815,A -85,B 0,C 180,E1 -20892.972,E2 -20892.972} C_VEL
LIN {X 0,Y 221.268,Z 418.965,A -85,B 0,C 180,E1 -20894.722,E2 -20894.722} C_VEL
LIN {X 0,Y 223.582,Z 418.605,A -85,B 0,C 180,E1 -20896.436,E2 -20896.436} C_VEL
LIN {X 0,Y 226.085,Z 417.714,A -85,B 0,C 180,E1 -20898.113,E2 -20898.113} C_VEL
